KUKA KRL program: EPS_2_25694_LG02_A_20260223033040.src

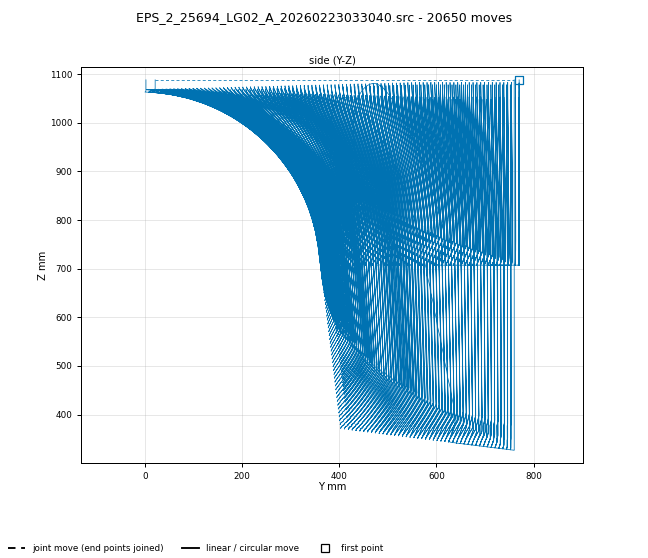
[picture p0: tool path of EPS_2_25694_LG02_A_20260223033040.src, 20650 of 20652 moves have a stored position in this frame; points joined in program order, loops and branches not executed]
&ACCESS RVP
&REL 4
&COMMENT QRS 19112012
&PARAM EDITMASK = *
DEF PART()
EXT BAS (BAS_COMMAND :IN,REAL :IN )
INT I
BAS (#INITMOV,0 )

;KUKA QRS Post kuka4.cps  Date:22-06-2017 !

File_ID=3059

QRS_PRE_INIT()

;Init var - Until changes are made in qrs_pre_init
Outlet_Square_prg=0
Inlet_1_Square_prg=0
Inlet_2_Square_prg=0
Inlet_3_Square_prg=0
Inlet_4_Square_prg=0
Inlet_5_Square_prg=0

Outlet_1={X 0.000, Y 562.000, Z 735.500, B 0.000, E1 0.000 }
Outlet_1={X 0.000, Y 562.000, Z 735.500, B 0.000, E1 0.000 }
Inlet_1={X 0.000, Y 562.000, Z 705.500, B 0.000, E1 182.000 }
Inlet_1={X 0.000, Y 562.000, Z 705.500, B 0.000, E1 182.000 }
Outlet_1_type=686
Inlet_1_type=686
Inlet_1_type=686
;QRS#1=Sidecore dimensions
;QRS#2=675-27" Concrete
;QRS#3=675-27" Concrete
;QRS#4=
;QRS#5=
;QRS#6=
;QRS#7=
;QRS#8=
;QRS#9=S306-38L
;QRS#10=S306-38L
;QRS#11=
;QRS#12=
;QRS#13=
;QRS#14=
;QRS#15=
;QRS#16=1524x152x1524 5'
;QRS#17=EPS Height
;QRS#18=1078,5
;QRS#19=*
;QRS#20= UPDATED VERSION 22-06-2017
;QRS#21=*
Outlet_Square=0550
Inlet_1_Square=0550
Inlet_2_Square=0
Inlet_3_Square=0
Inlet_4_Square=0
Inlet_5_Square=0
Mill_Square=1
Outlet_Square_Prg=265
Inlet_1_Square_prg=265
Inlet_1_Square_prg=265

QRS_INIT()

$ADVANCE=5

; T1
PTP {E1 171.77,E2 171.77}
PTP {X 0,Y 770.022,A -85,B 0,C 180,E1 171.77,E2 171.77,E3 0,E4 0,E5 0,E6 0}
QRS_SPEED_INIT()
LIN {X 0,Y 770.022,Z 1088.5,A -85,B 0,C 180,E1 171.77,E2 171.77,E3 0,E4 0,E5 0,E6 0} C_VEL
LIN {X 0,Y 770.022,Z 709.31,A -85,B 0,C 180,E1 171.77,E2 171.77} C_VEL
LIN {X 0,Y 769.965,Z 707.31,A -85,B 0,C 180,E1 171.919,E2 171.919} C_VEL
LIN {X 0,Y 770.089,Z 707.31,A -85,B 0,C 180,E1 175.346,E2 175.346} C_VEL
LIN {X 0,Y 770.137,Z 707.31,A -85,B 0,C 180,E1 180.93,E2 180.93} C_VEL
LIN {X 0,Y 770.147,Z 707.31,A -85,B 0,C 180,E1 186.522,E2 186.522} C_VEL
LIN {X 0,Y 770.143,Z 707.31,A -85,B 0,C 180,E1 190.282,E2 190.282} C_VEL
LIN {X 0,Y 769.943,Z 707.31,A -85,B 0,C 180,E1 194.091,E2 194.091} C_VEL
LIN {X 0,Y 769.516,Z 707.31,A -85,B 0,C 180,E1 196.027,E2 196.027} C_VEL
LIN {X 0,Y 770.012,Z 707.31,A -85,B 0,C 180,E1 199.927,E2 199.927} C_VEL
LIN {X 0,Y 769.316,Z 707.31,A -85,B 0,C 180,E1 202.191,E2 202.191} C_VEL
LIN {X 0,Y 769.398,Z 707.31,A -85,B 0,C 180,E1 203.958,E2 203.958} C_VEL
LIN {X 0,Y 769.902,Z 707.31,A -85,B 0,C 180,E1 205.993,E2 205.993} C_VEL
LIN {X 0,Y 769.961,Z 707.31,A -85,B 0,C 180,E1 210.209,E2 210.209} C_VEL
LIN {X 0,Y 770.093,Z 707.31,A -85,B 0,C 180,E1 210.674,E2 210.674} C_VEL
LIN {X 0,Y 769.97,Z 707.31,A -85,B 0,C 180,E1 214.616,E2 214.616} C_VEL
LIN {X 0,Y 769.539,Z 707.31,A -85,B 0,C 180,E1 217.274,E2 217.274} C_VEL
LIN {X 0,Y 769.964,Z 707.31,A -85,B 0,C 180,E1 219.272,E2 219.272} C_VEL
LIN {X 0,Y 769.757,Z 707.31,A -85,B 0,C 180,E1 220.266,E2 220.266} C_VEL
LIN {X 0,Y 769.848,Z 707.31,A -85,B 0,C 180,E1 224.269,E2 224.269} C_VEL
LIN {X 0,Y 769.688,Z 707.31,A -85,B 0,C 180,E1 225.72,E2 225.72} C_VEL
LIN {X 0,Y 769.829,Z 707.31,A -85,B 0,C 180,E1 229.727,E2 229.727} C_VEL
LIN {X 0,Y 769.876,Z 707.31,A -85,B 0,C 180,E1 230.723,E2 230.723} C_VEL
LIN {X 0,Y 769.499,Z 707.31,A -85,B 0,C 180,E1 233.066,E2 233.066} C_VEL
LIN {X 0,Y 769.922,Z 707.31,A -85,B 0,C 180,E1 235.382,E2 235.382} C_VEL
LIN {X 0,Y 770.114,Z 707.31,A -85,B 0,C 180,E1 240.252,E2 240.252} C_VEL
LIN {X 0,Y 769.925,Z 707.31,A -85,B 0,C 180,E1 240.47,E2 240.47} C_VEL
LIN {X 0,Y 768.498,Z 707.31,A -85,B 0,C 180,E1 240.635,E2 240.635} C_VEL
LIN {X 0,Y 768.109,Z 707.31,A -85,B 0,C 180,E1 240.658,E2 240.658} C_VEL
LIN {X 0,Y 769.095,Z 710.734,A -85,B 0,C 180,E1 240.752,E2 240.752} C_VEL
LIN {X 0,Y 769.603,Z 712.954,A -85,B 0,C 180,E1 240.796,E2 240.796} C_VEL
LIN {X 0,Y 769.831,Z 753.408,A -85,B 0,C 180,E1 241.229,E2 241.229} C_VEL
LIN {X 0,Y 769.934,Z 774.829,A -85,B 0,C 180,E1 241.5,E2 241.5} C_VEL
LIN {X 0,Y 769.745,Z 790.859,A -85,B 0,C 180,E1 241.76,E2 241.76} C_VEL
LIN {X 0,Y 769.973,Z 808.408,A -85,B 0,C 180,E1 242.135,E2 242.135} C_VEL
LIN {X 0,Y 769.941,Z 824.72,A -85,B 0,C 180,E1 242.54,E2 242.54} C_VEL
LIN {X 0,Y 769.833,Z 835.541,A -85,B 0,C 180,E1 242.844,E2 242.844} C_VEL
LIN {X 0,Y 769.948,Z 845.365,A -85,B 0,C 180,E1 243.157,E2 243.157} C_VEL
LIN {X 0,Y 769.988,Z 856.534,A -85,B 0,C 180,E1 243.531,E2 243.531} C_VEL
LIN {X 0,Y 769.881,Z 872.728,A -85,B 0,C 180,E1 244.138,E2 244.138} C_VEL
LIN {X 0,Y 770.005,Z 886.353,A -85,B 0,C 180,E1 244.711,E2 244.711} C_VEL
LIN {X 0,Y 769.999,Z 902.655,A -85,B 0,C 180,E1 245.473,E2 245.473} C_VEL
LIN {X 0,Y 769.936,Z 916.578,A -85,B 0,C 180,E1 246.187,E2 246.187} C_VEL
LIN {X 0,Y 769.972,Z 930.073,A -85,B 0,C 180,E1 246.948,E2 246.948} C_VEL
LIN {X 0,Y 770.004,Z 943.245,A -85,B 0,C 180,E1 247.759,E2 247.759} C_VEL
LIN {X 0,Y 770.023,Z 955.747,A -85,B 0,C 180,E1 248.596,E2 248.596} C_VEL
LIN {X 0,Y 769.988,Z 967.476,A -85,B 0,C 180,E1 249.447,E2 249.447} C_VEL
LIN {X 0,Y 769.996,Z 980.009,A -85,B 0,C 180,E1 250.443,E2 250.443} C_VEL
LIN {X 0,Y 770.035,Z 990.038,A -85,B 0,C 180,E1 251.305,E2 251.305} C_VEL
LIN {X 0,Y 769.912,Z 1001.083,A -85,B 0,C 180,E1 252.335,E2 252.335} C_VEL
LIN {X 0,Y 769.935,Z 1010.25,A -85,B 0,C 180,E1 253.265,E2 253.265} C_VEL
LIN {X 0,Y 770.052,Z 1020.333,A -85,B 0,C 180,E1 254.393,E2 254.393} C_VEL
LIN {X 0,Y 769.892,Z 1028.715,A -85,B 0,C 180,E1 255.404,E2 255.404} C_VEL
LIN {X 0,Y 769.938,Z 1037.752,A -85,B 0,C 180,E1 256.627,E2 256.627} C_VEL
LIN {X 0,Y 770.084,Z 1044.177,A -85,B 0,C 180,E1 257.583,E2 257.583} C_VEL
LIN {X 0,Y 769.904,Z 1051.422,A -85,B 0,C 180,E1 258.768,E2 258.768} C_VEL
LIN {X 0,Y 769.98,Z 1057.755,A -85,B 0,C 180,E1 259.952,E2 259.952} C_VEL
LIN {X 0,Y 770.017,Z 1062.183,A -85,B 0,C 180,E1 260.895,E2 260.895} C_VEL
LIN {X 0,Y 769.897,Z 1065.267,A -85,B 0,C 180,E1 261.6,E2 261.6} C_VEL
LIN {X 0,Y 769.889,Z 1069.496,A -85,B 0,C 180,E1 262.687,E2 262.687} C_VEL
LIN {X 0,Y 770.095,Z 1073.277,A -85,B 0,C 180,E1 263.852,E2 263.852} C_VEL
LIN {X 0,Y 769.943,Z 1075.349,A -85,B 0,C 180,E1 264.598,E2 264.598} C_VEL
LIN {X 0,Y 769.823,Z 1077.197,A -85,B 0,C 180,E1 265.344,E2 265.344} C_VEL
LIN {X 0,Y 769.892,Z 1079.406,A -85,B 0,C 180,E1 266.464,E2 266.464} C_VEL
LIN {X 0,Y 770.036,Z 1080.477,A -85,B 0,C 180,E1 267.209,E2 267.209} C_VEL
LIN {X 0,Y 769.896,Z 1081.687,A -85,B 0,C 180,E1 268.326,E2 268.326} C_VEL
LIN {X 0,Y 769.819,Z 1082.188,A -85,B 0,C 180,E1 269.07,E2 269.07} C_VEL
LIN {X 0,Y 770.094,Z 1082.112,A -85,B 0,C 180,E1 270.93,E2 270.93} C_VEL
LIN {X 0,Y 769.957,Z 1081.671,A -85,B 0,C 180,E1 271.674,E2 271.674} C_VEL
LIN {X 0,Y 769.922,Z 1080.508,A -85,B 0,C 180,E1 272.791,E2 272.791} C_VEL
LIN {X 0,Y 770.08,Z 1078.703,A -85,B 0,C 180,E1 273.908,E2 273.908} C_VEL
LIN {X 0,Y 769.95,Z 1077.164,A -85,B 0,C 180,E1 274.655,E2 274.655} C_VEL
LIN {X 0,Y 769.804,Z 1074.365,A -85,B 0,C 180,E1 275.777,E2 275.777} C_VEL
LIN {X 0,Y 769.869,Z 1072.15,A -85,B 0,C 180,E1 276.525,E2 276.525} C_VEL
LIN {X 0,Y 770.043,Z 1069.113,A -85,B 0,C 180,E1 277.415,E2 277.415} C_VEL
LIN {X 0,Y 769.819,Z 1063.335,A -85,B 0,C 180,E1 278.872,E2 278.872} C_VEL
LIN {X 0,Y 769.862,Z 1057.782,A -85,B 0,C 180,E1 280.05,E2 280.05} C_VEL
LIN {X 0,Y 770.061,Z 1051.388,A -85,B 0,C 180,E1 281.23,E2 281.23} C_VEL
LIN {X 0,Y 769.867,Z 1044.221,A -85,B 0,C 180,E1 282.42,E2 282.42} C_VEL
LIN {X 0,Y 769.93,Z 1036.081,A -85,B 0,C 180,E1 283.613,E2 283.613} C_VEL
LIN {X 0,Y 770.069,Z 1028.6,A -85,B 0,C 180,E1 284.603,E2 284.603} C_VEL
LIN {X 0,Y 769.93,Z 1018.062,A -85,B 0,C 180,E1 285.875,E2 285.875} C_VEL
LIN {X 0,Y 770.036,Z 1008.27,A -85,B 0,C 180,E1 286.937,E2 286.937} C_VEL
LIN {X 0,Y 770.027,Z 997.988,A -85,B 0,C 180,E1 287.96,E2 287.96} C_VEL
LIN {X 0,Y 769.959,Z 987.253,A -85,B 0,C 180,E1 288.942,E2 288.942} C_VEL
LIN {X 0,Y 770.039,Z 977.032,A -85,B 0,C 180,E1 289.803,E2 289.803} C_VEL
LIN {X 0,Y 770.021,Z 964.62,A -85,B 0,C 180,E1 290.763,E2 290.763} C_VEL
LIN {X 0,Y 769.992,Z 953.247,A -85,B 0,C 180,E1 291.577,E2 291.577} C_VEL
LIN {X 0,Y 770.022,Z 940.144,A -85,B 0,C 180,E1 292.436,E2 292.436} C_VEL
LIN {X 0,Y 770.026,Z 926.8,A -85,B 0,C 180,E1 293.24,E2 293.24} C_VEL
LIN {X 0,Y 769.999,Z 912.592,A -85,B 0,C 180,E1 294.022,E2 294.022} C_VEL
LIN {X 0,Y 769.954,Z 899.229,A -85,B 0,C 180,E1 294.697,E2 294.697} C_VEL
LIN {X 0,Y 770.006,Z 884.351,A -85,B 0,C 180,E1 295.375,E2 295.375} C_VEL
LIN {X 0,Y 769.96,Z 868.011,A -85,B 0,C 180,E1 296.044,E2 296.044} C_VEL
LIN {X 0,Y 769.9,Z 855.049,A -85,B 0,C 180,E1 296.527,E2 296.527} C_VEL
LIN {X 0,Y 769.996,Z 836.827,A -85,B 0,C 180,E1 297.113,E2 297.113} C_VEL
LIN {X 0,Y 769.884,Z 820.283,A -85,B 0,C 180,E1 297.579,E2 297.579} C_VEL
LIN {X 0,Y 769.807,Z 811.166,A -85,B 0,C 180,E1 297.804,E2 297.804} C_VEL
LIN {X 0,Y 769.928,Z 802.17,A -85,B 0,C 180,E1 298.003,E2 298.003} C_VEL
LIN {X 0,Y 769.948,Z 787.456,A -85,B 0,C 180,E1 298.293,E2 298.293} C_VEL
LIN {X 0,Y 769.698,Z 770.151,A -85,B 0,C 180,E1 298.575,E2 298.575} C_VEL
LIN {X 0,Y 769.766,Z 750.318,A -85,B 0,C 180,E1 298.806,E2 298.806} C_VEL
LIN {X 0,Y 769.682,Z 714.778,A -85,B 0,C 180,E1 299.181,E2 299.181} C_VEL
LIN {X 0,Y 769.131,Z 710.918,A -85,B 0,C 180,E1 299.245,E2 299.245} C_VEL
LIN {X 0,Y 767.905,Z 707.31,A -85,B 0,C 180,E1 299.334,E2 299.334} C_VEL
LIN {X 0,Y 769.925,Z 707.31,A -85,B 0,C 180,E1 299.53,E2 299.53} C_VEL
LIN {X 0,Y 770.155,Z 707.31,A -85,B 0,C 180,E1 299.746,E2 299.746} C_VEL
LIN {X 0,Y 770.109,Z 707.31,A -85,B 0,C 180,E1 300.676,E2 300.676} C_VEL
LIN {X 0,Y 769.956,Z 707.31,A -85,B 0,C 180,E1 304.616,E2 304.616} C_VEL
LIN {X 0,Y 769.531,Z 707.31,A -85,B 0,C 180,E1 307.274,E2 307.274} C_VEL
LIN {X 0,Y 769.966,Z 707.31,A -85,B 0,C 180,E1 309.271,E2 309.271} C_VEL
LIN {X 0,Y 769.769,Z 707.31,A -85,B 0,C 180,E1 310.267,E2 310.267} C_VEL
LIN {X 0,Y 769.861,Z 707.31,A -85,B 0,C 180,E1 314.268,E2 314.268} C_VEL
LIN {X 0,Y 769.694,Z 707.31,A -85,B 0,C 180,E1 315.72,E2 315.72} C_VEL
LIN {X 0,Y 769.828,Z 707.31,A -85,B 0,C 180,E1 319.727,E2 319.727} C_VEL
LIN {X 0,Y 769.883,Z 707.31,A -85,B 0,C 180,E1 320.723,E2 320.723} C_VEL
LIN {X 0,Y 769.518,Z 707.31,A -85,B 0,C 180,E1 323.067,E2 323.067} C_VEL
LIN {X 0,Y 769.966,Z 707.31,A -85,B 0,C 180,E1 325.384,E2 325.384} C_VEL
LIN {X 0,Y 770.084,Z 707.31,A -85,B 0,C 180,E1 329.327,E2 329.327} C_VEL
LIN {X 0,Y 769.954,Z 707.31,A -85,B 0,C 180,E1 329.791,E2 329.791} C_VEL
LIN {X 0,Y 769.909,Z 707.31,A -85,B 0,C 180,E1 334.007,E2 334.007} C_VEL
LIN {X 0,Y 769.391,Z 707.31,A -85,B 0,C 180,E1 336.042,E2 336.042} C_VEL
LIN {X 0,Y 769.371,Z 707.31,A -85,B 0,C 180,E1 338.063,E2 338.063} C_VEL
LIN {X 0,Y 770.006,Z 707.31,A -85,B 0,C 180,E1 340.073,E2 340.073} C_VEL
LIN {X 0,Y 769.528,Z 707.31,A -85,B 0,C 180,E1 343.974,E2 343.974} C_VEL
LIN {X 0,Y 769.936,Z 707.31,A -85,B 0,C 180,E1 345.909,E2 345.909} C_VEL
LIN {X 0,Y 770.137,Z 707.31,A -85,B 0,C 180,E1 349.718,E2 349.718} C_VEL
LIN {X 0,Y 770.151,Z 707.31,A -85,B 0,C 180,E1 353.478,E2 353.478} C_VEL
LIN {X 0,Y 770.123,Z 707.31,A -85,B 0,C 180,E1 359.07,E2 359.07} C_VEL
LIN {X 0,Y 770.092,Z 707.31,A -85,B 0,C 180,E1 364.654,E2 364.654} C_VEL
LIN {X 0,Y 770.054,Z 707.31,A -85,B 0,C 180,E1 370.283,E2 370.283} C_VEL
LIN {X 0,Y 769.882,Z 707.31,A -85,B 0,C 180,E1 374.092,E2 374.092} C_VEL
LIN {X 0,Y 769.483,Z 707.31,A -85,B 0,C 180,E1 376.027,E2 376.027} C_VEL
LIN {X 0,Y 770.04,Z 707.31,A -85,B 0,C 180,E1 379.926,E2 379.926} C_VEL
LIN {X 0,Y 769.697,Z 707.31,A -85,B 0,C 180,E1 382.261,E2 382.261} C_VEL
LIN {X 0,Y 770.058,Z 707.31,A -85,B 0,C 180,E1 383.936,E2 383.936} C_VEL
LIN {X 0,Y 769.305,Z 707.31,A -85,B 0,C 180,E1 386.69,E2 386.69} C_VEL
LIN {X 0,Y 769.438,Z 707.31,A -85,B 0,C 180,E1 388.1,E2 388.1} C_VEL
LIN {X 0,Y 769.806,Z 707.31,A -85,B 0,C 180,E1 390.216,E2 390.216} C_VEL
LIN {X 0,Y 769.886,Z 707.31,A -85,B 0,C 180,E1 394.62,E2 394.62} C_VEL
LIN {X 0,Y 769.484,Z 707.31,A -85,B 0,C 180,E1 397.269,E2 397.269} C_VEL
LIN {X 0,Y 769.902,Z 707.31,A -85,B 0,C 180,E1 399.275,E2 399.275} C_VEL
LIN {X 0,Y 769.868,Z 707.31,A -85,B 0,C 180,E1 400.276,E2 400.276} C_VEL
LIN {X 0,Y 769.855,Z 707.31,A -85,B 0,C 180,E1 404.268,E2 404.268} C_VEL
LIN {X 0,Y 769.692,Z 707.31,A -85,B 0,C 180,E1 405.72,E2 405.72} C_VEL
LIN {X 0,Y 769.873,Z 707.31,A -85,B 0,C 180,E1 409.724,E2 409.724} C_VEL
LIN {X 0,Y 770.006,Z 707.31,A -85,B 0,C 180,E1 410.731,E2 410.731} C_VEL
LIN {X 0,Y 769.993,Z 707.31,A -85,B 0,C 180,E1 413.093,E2 413.093} C_VEL
LIN {X 0,Y 769.36,Z 707.31,A -85,B 0,C 180,E1 415.936,E2 415.936} C_VEL
LIN {X 0,Y 770.019,Z 707.31,A -85,B 0,C 180,E1 418.367,E2 418.367} C_VEL
LIN {X 0,Y 769.919,Z 707.31,A -85,B 0,C 180,E1 418.779,E2 418.779} C_VEL
LIN {X 0,Y 768.954,Z 707.31,A -85,B 0,C 180,E1 418.939,E2 418.939} C_VEL
LIN {X 0,Y 768.758,Z 707.31,A -85,B 0,C 180,E1 418.958,E2 418.958} C_VEL
LIN {X 0,Y 768.921,Z 707.833,A -85,B 0,C 180,E1 418.984,E2 418.984} C_VEL
LIN {X 0,Y 769.552,Z 709.481,A -85,B 0,C 180,E1 419.027,E2 419.027} C_VEL
LIN {X 0,Y 769.707,Z 712.843,A -85,B 0,C 180,E1 419.068,E2 419.068} C_VEL
LIN {X 0,Y 769.864,Z 732.648,A -85,B 0,C 180,E1 419.294,E2 419.294} C_VEL
LIN {X 0,Y 769.85,Z 745.446,A -85,B 0,C 180,E1 419.462,E2 419.462} C_VEL
LIN {X 0,Y 769.757,Z 755.61,A -85,B 0,C 180,E1 419.624,E2 419.624} C_VEL
LIN {X 0,Y 769.862,Z 764.873,A -85,B 0,C 180,E1 419.801,E2 419.801} C_VEL
LIN {X 0,Y 769.858,Z 778.456,A -85,B 0,C 180,E1 420.086,E2 420.086} C_VEL
LIN {X 0,Y 769.821,Z 788.716,A -85,B 0,C 180,E1 420.335,E2 420.335} C_VEL
LIN {X 0,Y 769.911,Z 797.522,A -85,B 0,C 180,E1 420.574,E2 420.574} C_VEL
LIN {X 0,Y 769.941,Z 810.99,A -85,B 0,C 180,E1 420.968,E2 420.968} C_VEL
LIN {X 0,Y 769.825,Z 825.977,A -85,B 0,C 180,E1 421.459,E2 421.459} C_VEL
LIN {X 0,Y 769.962,Z 842.279,A -85,B 0,C 180,E1 422.077,E2 422.077} C_VEL
LIN {X 0,Y 769.92,Z 857.12,A -85,B 0,C 180,E1 422.698,E2 422.698} C_VEL
LIN {X 0,Y 769.996,Z 872.707,A -85,B 0,C 180,E1 423.43,E2 423.43} C_VEL
LIN {X 0,Y 770.001,Z 885.763,A -85,B 0,C 180,E1 424.099,E2 424.099} C_VEL
LIN {X 0,Y 769.962,Z 899.708,A -85,B 0,C 180,E1 424.881,E2 424.881} C_VEL
LIN {X 0,Y 769.97,Z 913.421,A -85,B 0,C 180,E1 425.725,E2 425.725} C_VEL
LIN {X 0,Y 769.995,Z 926.011,A -85,B 0,C 180,E1 426.57,E2 426.57} C_VEL
LIN {X 0,Y 770.041,Z 938.667,A -85,B 0,C 180,E1 427.497,E2 427.497} C_VEL
LIN {X 0,Y 769.962,Z 949.338,A -85,B 0,C 180,E1 428.34,E2 428.34} C_VEL
LIN {X 0,Y 769.965,Z 960.346,A -85,B 0,C 180,E1 429.286,E2 429.286} C_VEL
LIN {X 0,Y 770.061,Z 970.115,A -85,B 0,C 180,E1 430.198,E2 430.198} C_VEL
LIN {X 0,Y 769.912,Z 980.998,A -85,B 0,C 180,E1 431.302,E2 431.302} C_VEL
LIN {X 0,Y 769.954,Z 990.166,A -85,B 0,C 180,E1 432.323,E2 432.323} C_VEL
LIN {X 0,Y 770.03,Z 998.826,A -85,B 0,C 180,E1 433.38,E2 433.38} C_VEL
LIN {X 0,Y 769.876,Z 1007.704,A -85,B 0,C 180,E1 434.572,E2 434.572} C_VEL
LIN {X 0,Y 769.971,Z 1014.548,A -85,B 0,C 180,E1 435.59,E2 435.59} C_VEL
LIN {X 0,Y 770.061,Z 1019.352,A -85,B 0,C 180,E1 436.39,E2 436.39} C_VEL
LIN {X 0,Y 769.933,Z 1023.47,A -85,B 0,C 180,E1 437.104,E2 437.104} C_VEL
LIN {X 0,Y 769.882,Z 1028.518,A -85,B 0,C 180,E1 438.056,E2 438.056} C_VEL
LIN {X 0,Y 770.047,Z 1033.985,A -85,B 0,C 180,E1 439.244,E2 439.244} C_VEL
LIN {X 0,Y 769.897,Z 1037.803,A -85,B 0,C 180,E1 440.187,E2 440.187} C_VEL
LIN {X 0,Y 769.792,Z 1041.151,A -85,B 0,C 180,E1 441.128,E2 441.128} C_VEL
LIN {X 0,Y 769.817,Z 1042.735,A -85,B 0,C 180,E1 441.599,E2 441.599} C_VEL
LIN {X 0,Y 770.005,Z 1045.491,A -85,B 0,C 180,E1 442.611,E2 442.611} C_VEL
LIN {X 0,Y 769.973,Z 1047.526,A -85,B 0,C 180,E1 443.476,E2 443.476} C_VEL
LIN {X 0,Y 769.865,Z 1049.125,A -85,B 0,C 180,E1 444.224,E2 444.224} C_VEL
LIN {X 0,Y 769.912,Z 1050.786,A -85,B 0,C 180,E1 445.345,E2 445.345} C_VEL
LIN {X 0,Y 770.059,Z 1051.473,A -85,B 0,C 180,E1 446.092,E2 446.092} C_VEL
LIN {X 0,Y 769.847,Z 1052.232,A -85,B 0,C 180,E1 447.209,E2 447.209} C_VEL
LIN {X 0,Y 769.868,Z 1052.125,A -85,B 0,C 180,E1 449.07,E2 449.07} C_VEL
LIN {X 0,Y 770.051,Z 1051.152,A -85,B 0,C 180,E1 450.186,E2 450.186} C_VEL
LIN {X 0,Y 769.859,Z 1049.146,A -85,B 0,C 180,E1 451.674,E2 451.674} C_VEL
LIN {X 0,Y 769.988,Z 1046.777,A -85,B 0,C 180,E1 452.791,E2 452.791} C_VEL
LIN {X 0,Y 770.031,Z 1044.835,A -85,B 0,C 180,E1 453.536,E2 453.536} C_VEL
LIN {X 0,Y 769.875,Z 1042.817,A -85,B 0,C 180,E1 454.282,E2 454.282} C_VEL
LIN {X 0,Y 769.825,Z 1039.065,A -85,B 0,C 180,E1 455.403,E2 455.403} C_VEL
LIN {X 0,Y 770.076,Z 1033.466,A -85,B 0,C 180,E1 456.783,E2 456.783} C_VEL
LIN {X 0,Y 769.835,Z 1027.352,A -85,B 0,C 180,E1 458.086,E2 458.086} C_VEL
LIN {X 0,Y 769.838,Z 1021.898,A -85,B 0,C 180,E1 459.107,E2 459.107} C_VEL
LIN {X 0,Y 770.077,Z 1014.746,A -85,B 0,C 180,E1 460.283,E2 460.283} C_VEL
LIN {X 0,Y 769.892,Z 1006.814,A -85,B 0,C 180,E1 461.469,E2 461.469} C_VEL
LIN {X 0,Y 769.88,Z 997.877,A -85,B 0,C 180,E1 462.658,E2 462.658} C_VEL
LIN {X 0,Y 770.052,Z 987.84,A -85,B 0,C 180,E1 463.85,E2 463.85} C_VEL
LIN {X 0,Y 769.933,Z 979.058,A -85,B 0,C 180,E1 464.816,E2 464.816} C_VEL
LIN {X 0,Y 769.965,Z 967.997,A -85,B 0,C 180,E1 465.917,E2 465.917} C_VEL
LIN {X 0,Y 770.065,Z 958.104,A -85,B 0,C 180,E1 466.822,E2 466.822} C_VEL
LIN {X 0,Y 769.962,Z 946.275,A -85,B 0,C 180,E1 467.819,E2 467.819} C_VEL
LIN {X 0,Y 769.979,Z 934.941,A -85,B 0,C 180,E1 468.696,E2 468.696} C_VEL
LIN {X 0,Y 770.027,Z 922.862,A -85,B 0,C 180,E1 469.556,E2 469.556} C_VEL
LIN {X 0,Y 769.986,Z 910.109,A -85,B 0,C 180,E1 470.394,E2 470.394} C_VEL
LIN {X 0,Y 770.004,Z 897.682,A -85,B 0,C 180,E1 471.146,E2 471.146} C_VEL
LIN {X 0,Y 769.988,Z 883.743,A -85,B 0,C 180,E1 471.919,E2 471.919} C_VEL
LIN {X 0,Y 770.021,Z 869.346,A -85,B 0,C 180,E1 472.644,E2 472.644} C_VEL
LIN {X 0,Y 769.963,Z 853.47,A -85,B 0,C 180,E1 473.368,E2 473.368} C_VEL
LIN {X 0,Y 769.996,Z 838.489,A -85,B 0,C 180,E1 473.98,E2 473.98} C_VEL
LIN {X 0,Y 770.007,Z 823.517,A -85,B 0,C 180,E1 474.529,E2 474.529} C_VEL
LIN {X 0,Y 769.806,Z 806.359,A -85,B 0,C 180,E1 475.088,E2 475.088} C_VEL
LIN {X 0,Y 769.958,Z 790.171,A -85,B 0,C 180,E1 475.534,E2 475.534} C_VEL
LIN {X 0,Y 769.914,Z 773.708,A -85,B 0,C 180,E1 475.927,E2 475.927} C_VEL
LIN {X 0,Y 769.78,Z 761.942,A -85,B 0,C 180,E1 476.172,E2 476.172} C_VEL
LIN {X 0,Y 769.993,Z 742.231,A -85,B 0,C 180,E1 476.493,E2 476.493} C_VEL
LIN {X 0,Y 769.805,Z 720.28,A -85,B 0,C 180,E1 476.76,E2 476.76} C_VEL
LIN {X 0,Y 769.598,Z 707.31,A -85,B 0,C 180,E1 476.907,E2 476.907} C_VEL
LIN {X 0,Y 770.053,Z 707.31,A -85,B 0,C 180,E1 476.99,E2 476.99} C_VEL
LIN {X 0,Y 770.045,Z 707.31,A -85,B 0,C 180,E1 477.71,E2 477.71} C_VEL
LIN {X 0,Y 769.87,Z 707.31,A -85,B 0,C 180,E1 480.213,E2 480.213} C_VEL
LIN {X 0,Y 769.911,Z 707.31,A -85,B 0,C 180,E1 484.619,E2 484.619} C_VEL
LIN {X 0,Y 769.501,Z 707.31,A -85,B 0,C 180,E1 487.271,E2 487.271} C_VEL
LIN {X 0,Y 769.942,Z 707.31,A -85,B 0,C 180,E1 489.273,E2 489.273} C_VEL
LIN {X 0,Y 769.884,Z 707.31,A -85,B 0,C 180,E1 490.277,E2 490.277} C_VEL
LIN {X 0,Y 769.697,Z 707.31,A -85,B 0,C 180,E1 494.28,E2 494.28} C_VEL
LIN {X 0,Y 769.864,Z 707.31,A -85,B 0,C 180,E1 495.732,E2 495.732} C_VEL
LIN {X 0,Y 769.869,Z 707.31,A -85,B 0,C 180,E1 499.724,E2 499.724} C_VEL
LIN {X 0,Y 769.895,Z 707.31,A -85,B 0,C 180,E1 500.724,E2 500.724} C_VEL
LIN {X 0,Y 769.494,Z 707.31,A -85,B 0,C 180,E1 503.065,E2 503.065} C_VEL
LIN {X 0,Y 769.937,Z 707.31,A -85,B 0,C 180,E1 505.382,E2 505.382} C_VEL
LIN {X 0,Y 770.095,Z 707.31,A -85,B 0,C 180,E1 509.326,E2 509.326} C_VEL
LIN {X 0,Y 769.421,Z 707.31,A -85,B 0,C 180,E1 511.899,E2 511.899} C_VEL
LIN {X 0,Y 769.915,Z 707.31,A -85,B 0,C 180,E1 514.007,E2 514.007} C_VEL
LIN {X 0,Y 769.418,Z 707.31,A -85,B 0,C 180,E1 516.043,E2 516.043} C_VEL
LIN {X 0,Y 769.396,Z 707.31,A -85,B 0,C 180,E1 518.063,E2 518.063} C_VEL
LIN {X 0,Y 770.045,Z 707.31,A -85,B 0,C 180,E1 520.074,E2 520.074} C_VEL
LIN {X 0,Y 769.472,Z 707.31,A -85,B 0,C 180,E1 523.973,E2 523.973} C_VEL
LIN {X 0,Y 770.019,Z 707.31,A -85,B 0,C 180,E1 525.91,E2 525.91} C_VEL
LIN {X 0,Y 770.104,Z 707.31,A -85,B 0,C 180,E1 527.821,E2 527.821} C_VEL
LIN {X 0,Y 770.094,Z 707.31,A -85,B 0,C 180,E1 531.602,E2 531.602} C_VEL
LIN {X 0,Y 769.965,Z 707.31,A -85,B 0,C 180,E1 531.919,E2 531.919} C_VEL
LIN {X 0,Y 765.777,Z 707.31,A -85,B 0,C 180,E1 533.187,E2 533.187} C_VEL
LIN {X 0,Y 761.897,Z 707.31,A -85,B 0,C 180,E1 534.468,E2 534.468} C_VEL
LIN {X 0,Y 762.122,Z 707.31,A -85,B 0,C 180,E1 541.137,E2 541.137} C_VEL
LIN {X 0,Y 762.14,Z 707.31,A -85,B 0,C 180,E1 546.85,E2 546.85} C_VEL
LIN {X 0,Y 761.837,Z 707.31,A -85,B 0,C 180,E1 551.471,E2 551.471} C_VEL
LIN {X 0,Y 761.759,Z 707.31,A -85,B 0,C 180,E1 554.986,E2 554.986} C_VEL
LIN {X 0,Y 762.04,Z 707.31,A -85,B 0,C 180,E1 559.756,E2 559.756} C_VEL
LIN {X 0,Y 761.797,Z 707.31,A -85,B 0,C 180,E1 566.47,E2 566.47} C_VEL
LIN {X 0,Y 761.973,Z 707.31,A -85,B 0,C 180,E1 571.22,E2 571.22} C_VEL
LIN {X 0,Y 761.795,Z 707.31,A -85,B 0,C 180,E1 575.353,E2 575.353} C_VEL
LIN {X 0,Y 762.007,Z 707.31,A -85,B 0,C 180,E1 579.519,E2 579.519} C_VEL
LIN {X 0,Y 761.959,Z 707.31,A -85,B 0,C 180,E1 584.276,E2 584.276} C_VEL
LIN {X 0,Y 761.933,Z 707.31,A -85,B 0,C 180,E1 590.861,E2 590.861} C_VEL
LIN {X 0,Y 761.696,Z 707.31,A -85,B 0,C 180,E1 596.147,E2 596.147} C_VEL
LIN {X 0,Y 761.654,Z 707.31,A -85,B 0,C 180,E1 600.317,E2 600.317} C_VEL
LIN {X 0,Y 762.123,Z 712.337,A -85,B 0,C 180,E1 600.475,E2 600.475} C_VEL
LIN {X 0,Y 762.839,Z 786.85,A -85,B 0,C 180,E1 601.409,E2 601.409} C_VEL
LIN {X 0,Y 762.789,Z 832.67,A -85,B 0,C 180,E1 602.49,E2 602.49} C_VEL
LIN {X 0,Y 762.644,Z 876.024,A -85,B 0,C 180,E1 604.012,E2 604.012} C_VEL
LIN {X 0,Y 762.508,Z 917.78,A -85,B 0,C 180,E1 606.008,E2 606.008} C_VEL
LIN {X 0,Y 762.44,Z 956.472,A -85,B 0,C 180,E1 608.426,E2 608.426} C_VEL
LIN {X 0,Y 762.326,Z 990.608,A -85,B 0,C 180,E1 611.153,E2 611.153} C_VEL
LIN {X 0,Y 762.3,Z 1021.09,A -85,B 0,C 180,E1 614.284,E2 614.284} C_VEL
LIN {X 0,Y 762.278,Z 1046.013,A -85,B 0,C 180,E1 617.66,E2 617.66} C_VEL
LIN {X 0,Y 762.152,Z 1064.516,A -85,B 0,C 180,E1 621.135,E2 621.135} C_VEL
LIN {X 0,Y 762.179,Z 1075.63,A -85,B 0,C 180,E1 624.294,E2 624.294} C_VEL
LIN {X 0,Y 762.145,Z 1082.219,A -85,B 0,C 180,E1 627.72,E2 627.72} C_VEL
LIN {X 0,Y 762.233,Z 1083.17,A -85,B 0,C 180,E1 631.139,E2 631.139} C_VEL
LIN {X 0,Y 762.137,Z 1078.459,A -85,B 0,C 180,E1 634.561,E2 634.561} C_VEL
LIN {X 0,Y 762.103,Z 1068.014,A -85,B 0,C 180,E1 638,E2 638} C_VEL
LIN {X 0,Y 762.226,Z 1052.973,A -85,B 0,C 180,E1 641.177,E2 641.177} C_VEL
LIN {X 0,Y 762.303,Z 1029.54,A -85,B 0,C 180,E1 644.682,E2 644.682} C_VEL
LIN {X 0,Y 762.302,Z 1000.259,A -85,B 0,C 180,E1 647.945,E2 647.945} C_VEL
LIN {X 0,Y 762.412,Z 965.587,A -85,B 0,C 180,E1 650.91,E2 650.91} C_VEL
LIN {X 0,Y 762.559,Z 927.911,A -85,B 0,C 180,E1 653.418,E2 653.418} C_VEL
LIN {X 0,Y 762.713,Z 885.128,A -85,B 0,C 180,E1 655.603,E2 655.603} C_VEL
LIN {X 0,Y 762.881,Z 839.545,A -85,B 0,C 180,E1 657.305,E2 657.305} C_VEL
LIN {X 0,Y 762.975,Z 795.03,A -85,B 0,C 180,E1 658.428,E2 658.428} C_VEL
LIN {X 0,Y 762.839,Z 750.718,A -85,B 0,C 180,E1 659.089,E2 659.089} C_VEL
LIN {X 0,Y 762.065,Z 712.331,A -85,B 0,C 180,E1 659.527,E2 659.527} C_VEL
LIN {X 0,Y 761.246,Z 707.31,A -85,B 0,C 180,E1 659.651,E2 659.651} C_VEL
LIN {X 0,Y 762.267,Z 707.31,A -85,B 0,C 180,E1 659.801,E2 659.801} C_VEL
LIN {X 0,Y 761.798,Z 707.31,A -85,B 0,C 180,E1 665.359,E2 665.359} C_VEL
LIN {X 0,Y 762.009,Z 707.31,A -85,B 0,C 180,E1 669.522,E2 669.522} C_VEL
LIN {X 0,Y 761.973,Z 707.31,A -85,B 0,C 180,E1 674.282,E2 674.282} C_VEL
LIN {X 0,Y 761.939,Z 707.31,A -85,B 0,C 180,E1 680.864,E2 680.864} C_VEL
LIN {X 0,Y 761.801,Z 707.31,A -85,B 0,C 180,E1 686.155,E2 686.155} C_VEL
LIN {X 0,Y 761.889,Z 707.31,A -85,B 0,C 180,E1 690.185,E2 690.185} C_VEL
LIN {X 0,Y 761.983,Z 707.31,A -85,B 0,C 180,E1 694.056,E2 694.056} C_VEL
LIN {X 0,Y 762.007,Z 707.31,A -85,B 0,C 180,E1 700.243,E2 700.243} C_VEL
LIN {X 0,Y 761.957,Z 707.31,A -85,B 0,C 180,E1 706.195,E2 706.195} C_VEL
LIN {X 0,Y 761.898,Z 707.31,A -85,B 0,C 180,E1 710.846,E2 710.846} C_VEL
LIN {X 0,Y 761.786,Z 707.31,A -85,B 0,C 180,E1 714.294,E2 714.294} C_VEL
LIN {X 0,Y 762.089,Z 707.31,A -85,B 0,C 180,E1 718.863,E2 718.863} C_VEL
LIN {X 0,Y 762.146,Z 707.31,A -85,B 0,C 180,E1 724.564,E2 724.564} C_VEL
LIN {X 0,Y 762.151,Z 707.31,A -85,B 0,C 180,E1 730.31,E2 730.31} C_VEL
LIN {X 0,Y 761.701,Z 707.31,A -85,B 0,C 180,E1 734.991,E2 734.991} C_VEL
LIN {X 0,Y 761.885,Z 707.31,A -85,B 0,C 180,E1 740.8,E2 740.8} C_VEL
LIN {X 0,Y 761.782,Z 707.31,A -85,B 0,C 180,E1 744.695,E2 744.695} C_VEL
LIN {X 0,Y 761.782,Z 707.31,A -85,B 0,C 180,E1 749.825,E2 749.825} C_VEL
LIN {X 0,Y 761.721,Z 707.31,A -85,B 0,C 180,E1 755.347,E2 755.347} C_VEL
LIN {X 0,Y 762,Z 707.31,A -85,B 0,C 180,E1 759.525,E2 759.525} C_VEL
LIN {X 0,Y 761.967,Z 707.31,A -85,B 0,C 180,E1 764.278,E2 764.278} C_VEL
LIN {X 0,Y 762.079,Z 707.31,A -85,B 0,C 180,E1 770.854,E2 770.854} C_VEL
LIN {X 0,Y 761.514,Z 707.31,A -85,B 0,C 180,E1 774.754,E2 774.754} C_VEL
LIN {X 0,Y 761.814,Z 707.31,A -85,B 0,C 180,E1 778.68,E2 778.68} C_VEL
LIN {X 0,Y 762.938,Z 739.466,A -85,B 0,C 180,E1 779.094,E2 779.094} C_VEL
LIN {X 0,Y 762.785,Z 783.666,A -85,B 0,C 180,E1 779.934,E2 779.934} C_VEL
LIN {X 0,Y 762.625,Z 828.536,A -85,B 0,C 180,E1 781.285,E2 781.285} C_VEL
LIN {X 0,Y 762.657,Z 871.502,A -85,B 0,C 180,E1 783.116,E2 783.116} C_VEL
LIN {X 0,Y 762.44,Z 912.855,A -85,B 0,C 180,E1 785.455,E2 785.455} C_VEL
LIN {X 0,Y 762.334,Z 949.172,A -85,B 0,C 180,E1 788.117,E2 788.117} C_VEL
LIN {X 0,Y 762.191,Z 981.412,A -85,B 0,C 180,E1 791.151,E2 791.151} C_VEL
LIN {X 0,Y 762.1,Z 1007.099,A -85,B 0,C 180,E1 794.281,E2 794.281} C_VEL
LIN {X 0,Y 762.081,Z 1027.671,A -85,B 0,C 180,E1 797.658,E2 797.658} C_VEL
LIN {X 0,Y 762.005,Z 1041.297,A -85,B 0,C 180,E1 800.846,E2 800.846} C_VEL
LIN {X 0,Y 762.073,Z 1049.465,A -85,B 0,C 180,E1 803.872,E2 803.872} C_VEL
LIN {X 0,Y 762.126,Z 1053.024,A -85,B 0,C 180,E1 806.581,E2 806.581} C_VEL
LIN {X 0,Y 762.177,Z 1052.427,A -85,B 0,C 180,E1 810.001,E2 810.001} C_VEL
LIN {X 0,Y 762.21,Z 1046.286,A -85,B 0,C 180,E1 813.42,E2 813.42} C_VEL
LIN {X 0,Y 762.276,Z 1034.363,A -85,B 0,C 180,E1 816.851,E2 816.851} C_VEL
LIN {X 0,Y 762.275,Z 1015.941,A -85,B 0,C 180,E1 820.307,E2 820.307} C_VEL
LIN {X 0,Y 762.227,Z 991.64,A -85,B 0,C 180,E1 823.605,E2 823.605} C_VEL
LIN {X 0,Y 762.32,Z 962.721,A -85,B 0,C 180,E1 826.605,E2 826.605} C_VEL
LIN {X 0,Y 762.393,Z 929.673,A -85,B 0,C 180,E1 829.297,E2 829.297} C_VEL
LIN {X 0,Y 762.539,Z 893.05,A -85,B 0,C 180,E1 831.648,E2 831.648} C_VEL
LIN {X 0,Y 762.704,Z 852.297,A -85,B 0,C 180,E1 833.677,E2 833.677} C_VEL
LIN {X 0,Y 762.699,Z 807.525,A -85,B 0,C 180,E1 835.329,E2 835.329} C_VEL
LIN {X 0,Y 762.875,Z 759.589,A -85,B 0,C 180,E1 836.498,E2 836.498} C_VEL
LIN {X 0,Y 762.154,Z 707.31,A -85,B 0,C 180,E1 837.214,E2 837.214} C_VEL
LIN {X 0,Y 761.597,Z 707.31,A -85,B 0,C 180,E1 841.171,E2 841.171} C_VEL
LIN {X 0,Y 761.747,Z 707.31,A -85,B 0,C 180,E1 845.346,E2 845.346} C_VEL
LIN {X 0,Y 762.032,Z 707.31,A -85,B 0,C 180,E1 849.522,E2 849.522} C_VEL
LIN {X 0,Y 761.9,Z 707.31,A -85,B 0,C 180,E1 855.88,E2 855.88} C_VEL
LIN {X 0,Y 761.948,Z 707.31,A -85,B 0,C 180,E1 860.865,E2 860.865} C_VEL
LIN {X 0,Y 761.812,Z 707.31,A -85,B 0,C 180,E1 866.151,E2 866.151} C_VEL
LIN {X 0,Y 761.818,Z 707.31,A -85,B 0,C 180,E1 870.177,E2 870.177} C_VEL
LIN {X 0,Y 762.012,Z 707.31,A -85,B 0,C 180,E1 874.053,E2 874.053} C_VEL
LIN {X 0,Y 762.071,Z 707.31,A -85,B 0,C 180,E1 880.24,E2 880.24} C_VEL
LIN {X 0,Y 762.083,Z 707.31,A -85,B 0,C 180,E1 887,E2 887} C_VEL
LIN {X 0,Y 762.055,Z 707.31,A -85,B 0,C 180,E1 891.996,E2 891.996} C_VEL
LIN {X 0,Y 761.897,Z 707.31,A -85,B 0,C 180,E1 894.468,E2 894.468} C_VEL
LIN {X 0,Y 757.871,Z 707.31,A -85,B 0,C 180,E1 895.749,E2 895.749} C_VEL
LIN {X 0,Y 753.571,Z 707.31,A -85,B 0,C 180,E1 897.044,E2 897.044} C_VEL
LIN {X 0,Y 754.208,Z 707.31,A -85,B 0,C 180,E1 901.149,E2 901.149} C_VEL
LIN {X 0,Y 754.212,Z 707.31,A -85,B 0,C 180,E1 906.922,E2 906.922} C_VEL
LIN {X 0,Y 753.911,Z 707.31,A -85,B 0,C 180,E1 911.593,E2 911.593} C_VEL
LIN {X 0,Y 753.818,Z 707.31,A -85,B 0,C 180,E1 915.214,E2 915.214} C_VEL
LIN {X 0,Y 754.063,Z 707.31,A -85,B 0,C 180,E1 919.974,E2 919.974} C_VEL
LIN {X 0,Y 753.985,Z 707.31,A -85,B 0,C 180,E1 926.24,E2 926.24} C_VEL
LIN {X 0,Y 753.992,Z 707.31,A -85,B 0,C 180,E1 931.501,E2 931.501} C_VEL
LIN {X 0,Y 753.708,Z 707.31,A -85,B 0,C 180,E1 936.463,E2 936.463} C_VEL
LIN {X 0,Y 753.866,Z 707.31,A -85,B 0,C 180,E1 940.193,E2 940.193} C_VEL
LIN {X 0,Y 753.912,Z 707.31,A -85,B 0,C 180,E1 945.29,E2 945.29} C_VEL
LIN {X 0,Y 753.913,Z 707.31,A -85,B 0,C 180,E1 949.967,E2 949.967} C_VEL
LIN {X 0,Y 753.778,Z 707.31,A -85,B 0,C 180,E1 955.742,E2 955.742} C_VEL
LIN {X 0,Y 754.219,Z 707.31,A -85,B 0,C 180,E1 960.068,E2 960.068} C_VEL
LIN {X 0,Y 755.877,Z 722.616,A -85,B 0,C 180,E1 960.317,E2 960.317} C_VEL
LIN {X 0,Y 755.858,Z 789.553,A -85,B 0,C 180,E1 961.166,E2 961.166} C_VEL
LIN {X 0,Y 755.632,Z 838.054,A -85,B 0,C 180,E1 962.364,E2 962.364} C_VEL
LIN {X 0,Y 755.415,Z 885.307,A -85,B 0,C 180,E1 964.139,E2 964.139} C_VEL
LIN {X 0,Y 755.055,Z 929.178,A -85,B 0,C 180,E1 966.41,E2 966.41} C_VEL
LIN {X 0,Y 754.764,Z 967.337,A -85,B 0,C 180,E1 969.001,E2 969.001} C_VEL
LIN {X 0,Y 754.506,Z 1000.243,A -85,B 0,C 180,E1 971.861,E2 971.861} C_VEL
LIN {X 0,Y 754.31,Z 1029.534,A -85,B 0,C 180,E1 975.158,E2 975.158} C_VEL
LIN {X 0,Y 754.251,Z 1051.274,A -85,B 0,C 180,E1 978.409,E2 978.409} C_VEL
LIN {X 0,Y 754.205,Z 1066.858,A -85,B 0,C 180,E1 981.623,E2 981.623} C_VEL
LIN {X 0,Y 754.216,Z 1077.191,A -85,B 0,C 180,E1 984.812,E2 984.812} C_VEL
LIN {X 0,Y 754.241,Z 1082.219,A -85,B 0,C 180,E1 987.697,E2 987.697} C_VEL
LIN {X 0,Y 754.33,Z 1083.171,A -85,B 0,C 180,E1 991.151,E2 991.151} C_VEL
LIN {X 0,Y 754.228,Z 1078.459,A -85,B 0,C 180,E1 994.609,E2 994.609} C_VEL
LIN {X 0,Y 754.193,Z 1068.014,A -85,B 0,C 180,E1 998.085,E2 998.085} C_VEL
LIN {X 0,Y 754.347,Z 1052.974,A -85,B 0,C 180,E1 1001.295,E2 1001.295} C_VEL
LIN {X 0,Y 754.455,Z 1029.542,A -85,B 0,C 180,E1 1004.838,E2 1004.838} C_VEL
LIN {X 0,Y 754.575,Z 1000.254,A -85,B 0,C 180,E1 1008.136,E2 1008.136} C_VEL
LIN {X 0,Y 754.806,Z 965.588,A -85,B 0,C 180,E1 1011.131,E2 1011.131} C_VEL
LIN {X 0,Y 755.129,Z 927.914,A -85,B 0,C 180,E1 1013.663,E2 1013.663} C_VEL
LIN {X 0,Y 755.446,Z 885.349,A -85,B 0,C 180,E1 1015.858,E2 1015.858} C_VEL
LIN {X 0,Y 755.764,Z 840.029,A -85,B 0,C 180,E1 1017.568,E2 1017.568} C_VEL
LIN {X 0,Y 755.993,Z 795.724,A -85,B 0,C 180,E1 1018.7,E2 1018.7} C_VEL
LIN {X 0,Y 755.957,Z 752.369,A -85,B 0,C 180,E1 1019.362,E2 1019.362} C_VEL
LIN {X 0,Y 755.1,Z 714.015,A -85,B 0,C 180,E1 1019.809,E2 1019.809} C_VEL
LIN {X 0,Y 754.332,Z 707.31,A -85,B 0,C 180,E1 1019.968,E2 1019.968} C_VEL
LIN {X 0,Y 753.816,Z 707.31,A -85,B 0,C 180,E1 1025.66,E2 1025.66} C_VEL
LIN {X 0,Y 753.873,Z 707.31,A -85,B 0,C 180,E1 1030.199,E2 1030.199} C_VEL
LIN {X 0,Y 753.919,Z 707.31,A -85,B 0,C 180,E1 1035.294,E2 1035.294} C_VEL
LIN {X 0,Y 753.918,Z 707.31,A -85,B 0,C 180,E1 1039.972,E2 1039.972} C_VEL
LIN {X 0,Y 753.865,Z 707.31,A -85,B 0,C 180,E1 1045.75,E2 1045.75} C_VEL
LIN {X 0,Y 753.981,Z 707.31,A -85,B 0,C 180,E1 1049.84,E2 1049.84} C_VEL
LIN {X 0,Y 753.728,Z 707.31,A -85,B 0,C 180,E1 1055.028,E2 1055.028} C_VEL
LIN {X 0,Y 753.857,Z 707.31,A -85,B 0,C 180,E1 1060.871,E2 1060.871} C_VEL
LIN {X 0,Y 754.012,Z 707.31,A -85,B 0,C 180,E1 1066.047,E2 1066.047} C_VEL
LIN {X 0,Y 754.014,Z 707.31,A -85,B 0,C 180,E1 1070.75,E2 1070.75} C_VEL
LIN {X 0,Y 753.928,Z 707.31,A -85,B 0,C 180,E1 1074.234,E2 1074.234} C_VEL
LIN {X 0,Y 754.175,Z 707.31,A -85,B 0,C 180,E1 1078.851,E2 1078.851} C_VEL
LIN {X 0,Y 754.212,Z 707.31,A -85,B 0,C 180,E1 1084.612,E2 1084.612} C_VEL
LIN {X 0,Y 754.197,Z 707.31,A -85,B 0,C 180,E1 1090.42,E2 1090.42} C_VEL
LIN {X 0,Y 753.751,Z 707.31,A -85,B 0,C 180,E1 1095.2,E2 1095.2} C_VEL
LIN {X 0,Y 754.101,Z 707.31,A -85,B 0,C 180,E1 1099.978,E2 1099.978} C_VEL
LIN {X 0,Y 754.175,Z 707.31,A -85,B 0,C 180,E1 1103.697,E2 1103.697} C_VEL
LIN {X 0,Y 753.797,Z 707.31,A -85,B 0,C 180,E1 1110.181,E2 1110.181} C_VEL
LIN {X 0,Y 753.745,Z 707.31,A -85,B 0,C 180,E1 1115.667,E2 1115.667} C_VEL
LIN {X 0,Y 753.923,Z 707.31,A -85,B 0,C 180,E1 1120.2,E2 1120.2} C_VEL
LIN {X 0,Y 753.917,Z 707.31,A -85,B 0,C 180,E1 1125.291,E2 1125.291} C_VEL
LIN {X 0,Y 754.071,Z 707.31,A -85,B 0,C 180,E1 1131.608,E2 1131.608} C_VEL
LIN {X 0,Y 753.728,Z 707.31,A -85,B 0,C 180,E1 1137.123,E2 1137.123} C_VEL
LIN {X 0,Y 754.18,Z 707.31,A -85,B 0,C 180,E1 1138.351,E2 1138.351} C_VEL
LIN {X 0,Y 755.942,Z 718.996,A -85,B 0,C 180,E1 1138.557,E2 1138.557} C_VEL
LIN {X 0,Y 755.881,Z 765.457,A -85,B 0,C 180,E1 1139.245,E2 1139.245} C_VEL
LIN {X 0,Y 755.727,Z 809.818,A -85,B 0,C 180,E1 1140.379,E2 1140.379} C_VEL
LIN {X 0,Y 755.407,Z 854.961,A -85,B 0,C 180,E1 1142.079,E2 1142.079} C_VEL
LIN {X 0,Y 755.085,Z 898.214,A -85,B 0,C 180,E1 1144.308,E2 1144.308} C_VEL
LIN {X 0,Y 754.814,Z 937.295,A -85,B 0,C 180,E1 1146.954,E2 1146.954} C_VEL
LIN {X 0,Y 754.585,Z 971.141,A -85,B 0,C 180,E1 1149.91,E2 1149.91} C_VEL
LIN {X 0,Y 754.438,Z 999.469,A -85,B 0,C 180,E1 1153.107,E2 1153.107} C_VEL
LIN {X 0,Y 754.332,Z 1022.918,A -85,B 0,C 180,E1 1156.649,E2 1156.649} C_VEL
LIN {X 0,Y 754.212,Z 1038.2,A -85,B 0,C 180,E1 1159.917,E2 1159.917} C_VEL
LIN {X 0,Y 754.282,Z 1047.899,A -85,B 0,C 180,E1 1163.077,E2 1163.077} C_VEL
LIN {X 0,Y 754.225,Z 1053.005,A -85,B 0,C 180,E1 1166.545,E2 1166.545} C_VEL
LIN {X 0,Y 754.277,Z 1052.446,A -85,B 0,C 180,E1 1170.001,E2 1170.001} C_VEL
LIN {X 0,Y 754.334,Z 1046.344,A -85,B 0,C 180,E1 1173.456,E2 1173.456} C_VEL
LIN {X 0,Y 754.363,Z 1034.464,A -85,B 0,C 180,E1 1176.923,E2 1176.923} C_VEL
LIN {X 0,Y 754.404,Z 1016.075,A -85,B 0,C 180,E1 1180.416,E2 1180.416} C_VEL
LIN {X 0,Y 754.437,Z 991.833,A -85,B 0,C 180,E1 1183.748,E2 1183.748} C_VEL
LIN {X 0,Y 754.616,Z 963.246,A -85,B 0,C 180,E1 1186.753,E2 1186.753} C_VEL
LIN {X 0,Y 754.825,Z 930.606,A -85,B 0,C 180,E1 1189.453,E2 1189.453} C_VEL
LIN {X 0,Y 755.123,Z 893.467,A -85,B 0,C 180,E1 1191.871,E2 1191.871} C_VEL
LIN {X 0,Y 755.438,Z 852.955,A -85,B 0,C 180,E1 1193.915,E2 1193.915} C_VEL
LIN {X 0,Y 755.602,Z 807.775,A -85,B 0,C 180,E1 1195.601,E2 1195.601} C_VEL
LIN {X 0,Y 755.895,Z 760.769,A -85,B 0,C 180,E1 1196.762,E2 1196.762} C_VEL
LIN {X 0,Y 755.113,Z 710.992,A -85,B 0,C 180,E1 1197.474,E2 1197.474} C_VEL
LIN {X 0,Y 754.145,Z 707.31,A -85,B 0,C 180,E1 1197.606,E2 1197.606} C_VEL
LIN {X 0,Y 753.593,Z 707.31,A -85,B 0,C 180,E1 1202.885,E2 1202.885} C_VEL
LIN {X 0,Y 753.7,Z 707.31,A -85,B 0,C 180,E1 1207.099,E2 1207.099} C_VEL
LIN {X 0,Y 753.62,Z 707.31,A -85,B 0,C 180,E1 1211.574,E2 1211.574} C_VEL
LIN {X 0,Y 753.836,Z 707.31,A -85,B 0,C 180,E1 1216.361,E2 1216.361} C_VEL
LIN {X 0,Y 753.839,Z 707.31,A -85,B 0,C 180,E1 1221.629,E2 1221.629} C_VEL
LIN {X 0,Y 753.862,Z 707.31,A -85,B 0,C 180,E1 1225.745,E2 1225.745} C_VEL
LIN {X 0,Y 753.94,Z 707.31,A -85,B 0,C 180,E1 1229.833,E2 1229.833} C_VEL
LIN {X 0,Y 753.772,Z 707.31,A -85,B 0,C 180,E1 1235.025,E2 1235.025} C_VEL
LIN {X 0,Y 753.857,Z 707.31,A -85,B 0,C 180,E1 1240.874,E2 1240.874} C_VEL
LIN {X 0,Y 754.21,Z 707.31,A -85,B 0,C 180,E1 1247.229,E2 1247.229} C_VEL
LIN {X 0,Y 754.137,Z 707.31,A -85,B 0,C 180,E1 1251.914,E2 1251.914} C_VEL
LIN {X 0,Y 753.738,Z 707.31,A -85,B 0,C 180,E1 1256.54,E2 1256.54} C_VEL
LIN {X 0,Y 753.571,Z 707.31,A -85,B 0,C 180,E1 1257.044,E2 1257.044} C_VEL
LIN {X 0,Y 749.478,Z 707.31,A -85,B 0,C 180,E1 1258.341,E2 1258.341} C_VEL
LIN {X 0,Y 745.8,Z 707.31,A -85,B 0,C 180,E1 1259.652,E2 1259.652} C_VEL
LIN {X 0,Y 745.783,Z 707.31,A -85,B 0,C 180,E1 1262.327,E2 1262.327} C_VEL
LIN {X 0,Y 746.29,Z 707.31,A -85,B 0,C 180,E1 1266.996,E2 1266.996} C_VEL
LIN {X 0,Y 745.989,Z 707.31,A -85,B 0,C 180,E1 1271.718,E2 1271.718} C_VEL
LIN {X 0,Y 745.91,Z 707.31,A -85,B 0,C 180,E1 1275.312,E2 1275.312} C_VEL
LIN {X 0,Y 745.868,Z 707.31,A -85,B 0,C 180,E1 1280.836,E2 1280.836} C_VEL
LIN {X 0,Y 745.966,Z 707.31,A -85,B 0,C 180,E1 1286.639,E2 1286.639} C_VEL
LIN {X 0,Y 746.011,Z 707.31,A -85,B 0,C 180,E1 1291.877,E2 1291.877} C_VEL
LIN {X 0,Y 745.839,Z 707.31,A -85,B 0,C 180,E1 1296.099,E2 1296.099} C_VEL
LIN {X 0,Y 745.861,Z 707.31,A -85,B 0,C 180,E1 1300.55,E2 1300.55} C_VEL
LIN {X 0,Y 746.004,Z 707.31,A -85,B 0,C 180,E1 1305.311,E2 1305.311} C_VEL
LIN {X 0,Y 745.91,Z 707.31,A -85,B 0,C 180,E1 1310.964,E2 1310.964} C_VEL
LIN {X 0,Y 745.888,Z 707.31,A -85,B 0,C 180,E1 1315.328,E2 1315.328} C_VEL
LIN {X 0,Y 746.211,Z 708.049,A -85,B 0,C 180,E1 1319.734,E2 1319.734} C_VEL
LIN {X 0,Y 749.027,Z 721.889,A -85,B 0,C 180,E1 1320.01,E2 1320.01} C_VEL
LIN {X 0,Y 748.931,Z 789.558,A -85,B 0,C 180,E1 1320.874,E2 1320.874} C_VEL
LIN {X 0,Y 748.562,Z 838.058,A -85,B 0,C 180,E1 1322.08,E2 1322.08} C_VEL
LIN {X 0,Y 748.149,Z 884.93,A -85,B 0,C 180,E1 1323.853,E2 1323.853} C_VEL
LIN {X 0,Y 747.628,Z 927.895,A -85,B 0,C 180,E1 1326.084,E2 1326.084} C_VEL
LIN {X 0,Y 747.163,Z 967.678,A -85,B 0,C 180,E1 1328.805,E2 1328.805} C_VEL
LIN {X 0,Y 746.806,Z 1000.244,A -85,B 0,C 180,E1 1331.667,E2 1331.667} C_VEL
LIN {X 0,Y 746.516,Z 1029.535,A -85,B 0,C 180,E1 1334.999,E2 1334.999} C_VEL
LIN {X 0,Y 746.391,Z 1051.275,A -85,B 0,C 180,E1 1338.285,E2 1338.285} C_VEL
LIN {X 0,Y 746.341,Z 1066.859,A -85,B 0,C 180,E1 1341.534,E2 1341.534} C_VEL
LIN {X 0,Y 746.321,Z 1077.191,A -85,B 0,C 180,E1 1344.757,E2 1344.757} C_VEL
LIN {X 0,Y 746.338,Z 1082.219,A -85,B 0,C 180,E1 1347.672,E2 1347.672} C_VEL
LIN {X 0,Y 746.427,Z 1083.171,A -85,B 0,C 180,E1 1351.163,E2 1351.163} C_VEL
LIN {X 0,Y 746.322,Z 1078.46,A -85,B 0,C 180,E1 1354.658,E2 1354.658} C_VEL
LIN {X 0,Y 746.346,Z 1069.166,A -85,B 0,C 180,E1 1357.877,E2 1357.877} C_VEL
LIN {X 0,Y 746.493,Z 1052.975,A -85,B 0,C 180,E1 1361.415,E2 1361.415} C_VEL
LIN {X 0,Y 746.609,Z 1029.543,A -85,B 0,C 180,E1 1364.998,E2 1364.998} C_VEL
LIN {X 0,Y 746.859,Z 1000.255,A -85,B 0,C 180,E1 1368.33,E2 1368.33} C_VEL
LIN {X 0,Y 747.215,Z 966.286,A -85,B 0,C 180,E1 1371.304,E2 1371.304} C_VEL
LIN {X 0,Y 747.67,Z 927.917,A -85,B 0,C 180,E1 1373.913,E2 1373.913} C_VEL
LIN {X 0,Y 748.194,Z 884.961,A -85,B 0,C 180,E1 1376.144,E2 1376.144} C_VEL
LIN {X 0,Y 748.644,Z 841.607,A -85,B 0,C 180,E1 1377.799,E2 1377.799} C_VEL
LIN {X 0,Y 748.995,Z 799.12,A -85,B 0,C 180,E1 1378.922,E2 1378.922} C_VEL
LIN {X 0,Y 749.086,Z 754.307,A -85,B 0,C 180,E1 1379.637,E2 1379.637} C_VEL
LIN {X 0,Y 748.377,Z 716.318,A -85,B 0,C 180,E1 1380.079,E2 1380.079} C_VEL
LIN {X 0,Y 746.349,Z 707.31,A -85,B 0,C 180,E1 1380.295,E2 1380.295} C_VEL
LIN {X 0,Y 745.835,Z 707.31,A -85,B 0,C 180,E1 1386.101,E2 1386.101} C_VEL
LIN {X 0,Y 745.873,Z 707.31,A -85,B 0,C 180,E1 1390.552,E2 1390.552} C_VEL
LIN {X 0,Y 746.012,Z 707.31,A -85,B 0,C 180,E1 1395.313,E2 1395.313} C_VEL
LIN {X 0,Y 745.919,Z 707.31,A -85,B 0,C 180,E1 1400.969,E2 1400.969} C_VEL
LIN {X 0,Y 745.894,Z 707.31,A -85,B 0,C 180,E1 1406.405,E2 1406.405} C_VEL
LIN {X 0,Y 745.821,Z 707.31,A -85,B 0,C 180,E1 1410.89,E2 1410.89} C_VEL
LIN {X 0,Y 745.935,Z 707.31,A -85,B 0,C 180,E1 1414.749,E2 1414.749} C_VEL
LIN {X 0,Y 746.059,Z 707.31,A -85,B 0,C 180,E1 1419.802,E2 1419.802} C_VEL
LIN {X 0,Y 746.068,Z 707.31,A -85,B 0,C 180,E1 1425.895,E2 1425.895} C_VEL
LIN {X 0,Y 746.148,Z 707.31,A -85,B 0,C 180,E1 1430.652,E2 1430.652} C_VEL
LIN {X 0,Y 745.908,Z 707.31,A -85,B 0,C 180,E1 1434.551,E2 1434.551} C_VEL
LIN {X 0,Y 746.262,Z 707.31,A -85,B 0,C 180,E1 1438.839,E2 1438.839} C_VEL
LIN {X 0,Y 745.946,Z 707.31,A -85,B 0,C 180,E1 1445.48,E2 1445.48} C_VEL
LIN {X 0,Y 746.244,Z 707.31,A -85,B 0,C 180,E1 1450.533,E2 1450.533} C_VEL
LIN {X 0,Y 745.844,Z 707.31,A -85,B 0,C 180,E1 1455.317,E2 1455.317} C_VEL
LIN {X 0,Y 746.044,Z 707.31,A -85,B 0,C 180,E1 1460.875,E2 1460.875} C_VEL
LIN {X 0,Y 745.81,Z 707.31,A -85,B 0,C 180,E1 1465.26,E2 1465.26} C_VEL
LIN {X 0,Y 745.833,Z 707.31,A -85,B 0,C 180,E1 1470.53,E2 1470.53} C_VEL
LIN {X 0,Y 745.778,Z 707.31,A -85,B 0,C 180,E1 1476.107,E2 1476.107} C_VEL
LIN {X 0,Y 745.929,Z 707.31,A -85,B 0,C 180,E1 1480.551,E2 1480.551} C_VEL
LIN {X 0,Y 746.007,Z 707.31,A -85,B 0,C 180,E1 1485.316,E2 1485.316} C_VEL
LIN {X 0,Y 746.09,Z 707.31,A -85,B 0,C 180,E1 1490.977,E2 1490.977} C_VEL
LIN {X 0,Y 745.669,Z 707.31,A -85,B 0,C 180,E1 1495.318,E2 1495.318} C_VEL
LIN {X 0,Y 746.195,Z 707.31,A -85,B 0,C 180,E1 1498.002,E2 1498.002} C_VEL
LIN {X 0,Y 749.026,Z 716.059,A -85,B 0,C 180,E1 1498.226,E2 1498.226} C_VEL
LIN {X 0,Y 748.911,Z 765.18,A -85,B 0,C 180,E1 1498.946,E2 1498.946} C_VEL
LIN {X 0,Y 748.631,Z 809.987,A -85,B 0,C 180,E1 1500.101,E2 1500.101} C_VEL
LIN {X 0,Y 748.157,Z 853.676,A -85,B 0,C 180,E1 1501.754,E2 1501.754} C_VEL
LIN {X 0,Y 747.656,Z 895.833,A -85,B 0,C 180,E1 1503.921,E2 1503.921} C_VEL
LIN {X 0,Y 747.201,Z 933.827,A -85,B 0,C 180,E1 1506.467,E2 1506.467} C_VEL
LIN {X 0,Y 746.845,Z 967.913,A -85,B 0,C 180,E1 1509.399,E2 1509.399} C_VEL
LIN {X 0,Y 746.558,Z 996.446,A -85,B 0,C 180,E1 1512.564,E2 1512.564} C_VEL
LIN {X 0,Y 746.452,Z 1017.497,A -85,B 0,C 180,E1 1515.6,E2 1515.6} C_VEL
LIN {X 0,Y 746.431,Z 1034.417,A -85,B 0,C 180,E1 1518.88,E2 1518.88} C_VEL
LIN {X 0,Y 746.382,Z 1046.402,A -85,B 0,C 180,E1 1522.417,E2 1522.417} C_VEL
LIN {X 0,Y 746.297,Z 1051.936,A -85,B 0,C 180,E1 1525.342,E2 1525.342} C_VEL
LIN {X 0,Y 746.214,Z 1053.252,A -85,B 0,C 180,E1 1528.837,E2 1528.837} C_VEL
LIN {X 0,Y 746.274,Z 1049.047,A -85,B 0,C 180,E1 1532.328,E2 1532.328} C_VEL
LIN {X 0,Y 746.262,Z 1039.185,A -85,B 0,C 180,E1 1535.828,E2 1535.828} C_VEL
LIN {X 0,Y 746.28,Z 1024.636,A -85,B 0,C 180,E1 1539.055,E2 1539.055} C_VEL
LIN {X 0,Y 746.423,Z 1005.359,A -85,B 0,C 180,E1 1542.16,E2 1542.16} C_VEL
LIN {X 0,Y 746.695,Z 979.799,A -85,B 0,C 180,E1 1545.298,E2 1545.298} C_VEL
LIN {X 0,Y 747.02,Z 947.897,A -85,B 0,C 180,E1 1548.327,E2 1548.327} C_VEL
LIN {X 0,Y 747.482,Z 910.148,A -85,B 0,C 180,E1 1551.106,E2 1551.106} C_VEL
LIN {X 0,Y 748.042,Z 869.234,A -85,B 0,C 180,E1 1553.427,E2 1553.427} C_VEL
LIN {X 0,Y 748.546,Z 824.817,A -85,B 0,C 180,E1 1555.309,E2 1555.309} C_VEL
LIN {X 0,Y 748.869,Z 780.176,A -85,B 0,C 180,E1 1556.633,E2 1556.633} C_VEL
LIN {X 0,Y 749.188,Z 736.743,A -85,B 0,C 180,E1 1557.432,E2 1557.432} C_VEL
LIN {X 0,Y 748.27,Z 713.356,A -85,B 0,C 180,E1 1557.746,E2 1557.746} C_VEL
LIN {X 0,Y 746.195,Z 707.31,A -85,B 0,C 180,E1 1557.925,E2 1557.925} C_VEL
LIN {X 0,Y 745.752,Z 707.31,A -85,B 0,C 180,E1 1563.575,E2 1563.575} C_VEL
LIN {X 0,Y 745.965,Z 707.31,A -85,B 0,C 180,E1 1569.033,E2 1569.033} C_VEL
LIN {X 0,Y 746.081,Z 707.31,A -85,B 0,C 180,E1 1575.309,E2 1575.309} C_VEL
LIN {X 0,Y 745.933,Z 707.31,A -85,B 0,C 180,E1 1580.964,E2 1580.964} C_VEL
LIN {X 0,Y 745.887,Z 707.31,A -85,B 0,C 180,E1 1586.408,E2 1586.408} C_VEL
LIN {X 0,Y 745.812,Z 707.31,A -85,B 0,C 180,E1 1590.893,E2 1590.893} C_VEL
LIN {X 0,Y 745.975,Z 707.31,A -85,B 0,C 180,E1 1594.746,E2 1594.746} C_VEL
LIN {X 0,Y 746.101,Z 707.31,A -85,B 0,C 180,E1 1599.799,E2 1599.799} C_VEL
LIN {X 0,Y 746.171,Z 707.31,A -85,B 0,C 180,E1 1605.892,E2 1605.892} C_VEL
LIN {X 0,Y 746.123,Z 707.31,A -85,B 0,C 180,E1 1610.647,E2 1610.647} C_VEL
LIN {X 0,Y 746.289,Z 707.31,A -85,B 0,C 180,E1 1615.339,E2 1615.339} C_VEL
LIN {X 0,Y 745.8,Z 707.31,A -85,B 0,C 180,E1 1619.652,E2 1619.652} C_VEL
LIN {X 0,Y 742.083,Z 707.31,A -85,B 0,C 180,E1 1620.971,E2 1620.971} C_VEL
LIN {X 0,Y 737.912,Z 707.31,A -85,B 0,C 180,E1 1622.304,E2 1622.304} C_VEL
LIN {X 0,Y 738.364,Z 707.31,A -85,B 0,C 180,E1 1627.071,E2 1627.071} C_VEL
LIN {X 0,Y 738.079,Z 707.31,A -85,B 0,C 180,E1 1631.846,E2 1631.846} C_VEL
LIN {X 0,Y 737.989,Z 707.31,A -85,B 0,C 180,E1 1635.48,E2 1635.48} C_VEL
LIN {X 0,Y 738.096,Z 707.31,A -85,B 0,C 180,E1 1640.425,E2 1640.425} C_VEL
LIN {X 0,Y 738.035,Z 707.31,A -85,B 0,C 180,E1 1645.54,E2 1645.54} C_VEL
LIN {X 0,Y 738.178,Z 707.31,A -85,B 0,C 180,E1 1650.876,E2 1650.876} C_VEL
LIN {X 0,Y 738.032,Z 707.31,A -85,B 0,C 180,E1 1655.091,E2 1655.091} C_VEL
LIN {X 0,Y 737.978,Z 707.31,A -85,B 0,C 180,E1 1660.555,E2 1660.555} C_VEL
LIN {X 0,Y 737.966,Z 707.31,A -85,B 0,C 180,E1 1665.945,E2 1665.945} C_VEL
LIN {X 0,Y 737.961,Z 707.31,A -85,B 0,C 180,E1 1671.286,E2 1671.286} C_VEL
LIN {X 0,Y 737.857,Z 707.31,A -85,B 0,C 180,E1 1676.322,E2 1676.322} C_VEL
LIN {X 0,Y 738.102,Z 707.31,A -85,B 0,C 180,E1 1679.342,E2 1679.342} C_VEL
LIN {X 0,Y 742.131,Z 719.663,A -85,B 0,C 180,E1 1679.678,E2 1679.678} C_VEL
LIN {X 0,Y 742.015,Z 789.558,A -85,B 0,C 180,E1 1680.576,E2 1680.576} C_VEL
LIN {X 0,Y 741.505,Z 838.384,A -85,B 0,C 180,E1 1681.801,E2 1681.801} C_VEL
LIN {X 0,Y 740.902,Z 885.4,A -85,B 0,C 180,E1 1683.598,E2 1683.598} C_VEL
LIN {X 0,Y 740.192,Z 929.201,A -85,B 0,C 180,E1 1685.909,E2 1685.909} C_VEL
LIN {X 0,Y 739.609,Z 966.936,A -85,B 0,C 180,E1 1688.517,E2 1688.517} C_VEL
LIN {X 0,Y 739.102,Z 1000.245,A -85,B 0,C 180,E1 1691.47,E2 1691.47} C_VEL
LIN {X 0,Y 738.751,Z 1028.405,A -85,B 0,C 180,E1 1694.689,E2 1694.689} C_VEL
LIN {X 0,Y 738.541,Z 1051.277,A -85,B 0,C 180,E1 1698.159,E2 1698.159} C_VEL
LIN {X 0,Y 738.453,Z 1066.859,A -85,B 0,C 180,E1 1701.443,E2 1701.443} C_VEL
LIN {X 0,Y 738.412,Z 1077.444,A -85,B 0,C 180,E1 1704.799,E2 1704.799} C_VEL
LIN {X 0,Y 738.46,Z 1082.22,A -85,B 0,C 180,E1 1707.647,E2 1707.647} C_VEL
LIN {X 0,Y 738.524,Z 1083.17,A -85,B 0,C 180,E1 1711.175,E2 1711.175} C_VEL
LIN {X 0,Y 738.443,Z 1078.46,A -85,B 0,C 180,E1 1714.708,E2 1714.708} C_VEL
LIN {X 0,Y 738.458,Z 1069.166,A -85,B 0,C 180,E1 1717.962,E2 1717.962} C_VEL
LIN {X 0,Y 738.617,Z 1052.976,A -85,B 0,C 180,E1 1721.539,E2 1721.539} C_VEL
LIN {X 0,Y 738.802,Z 1029.767,A -85,B 0,C 180,E1 1725.129,E2 1725.129} C_VEL
LIN {X 0,Y 739.108,Z 1000.256,A -85,B 0,C 180,E1 1728.529,E2 1728.529} C_VEL
LIN {X 0,Y 739.627,Z 965.878,A -85,B 0,C 180,E1 1731.564,E2 1731.564} C_VEL
LIN {X 0,Y 740.283,Z 926.516,A -85,B 0,C 180,E1 1734.249,E2 1734.249} C_VEL
LIN {X 0,Y 740.981,Z 884.496,A -85,B 0,C 180,E1 1736.439,E2 1736.439} C_VEL
LIN {X 0,Y 741.618,Z 839.844,A -85,B 0,C 180,E1 1738.146,E2 1738.146} C_VEL
LIN {X 0,Y 742.071,Z 796.107,A -85,B 0,C 180,E1 1739.282,E2 1739.282} C_VEL
LIN {X 0,Y 742.225,Z 753.719,A -85,B 0,C 180,E1 1739.945,E2 1739.945} C_VEL
LIN {X 0,Y 741.663,Z 718.409,A -85,B 0,C 180,E1 1740.357,E2 1740.357} C_VEL
LIN {X 0,Y 738.364,Z 707.31,A -85,B 0,C 180,E1 1740.655,E2 1740.655} C_VEL
LIN {X 0,Y 738.032,Z 707.31,A -85,B 0,C 180,E1 1745.094,E2 1745.094} C_VEL
LIN {X 0,Y 737.988,Z 707.31,A -85,B 0,C 180,E1 1750.561,E2 1750.561} C_VEL
LIN {X 0,Y 737.971,Z 707.31,A -85,B 0,C 180,E1 1755.948,E2 1755.948} C_VEL
LIN {X 0,Y 737.974,Z 707.31,A -85,B 0,C 180,E1 1761.288,E2 1761.288} C_VEL
LIN {X 0,Y 737.991,Z 707.31,A -85,B 0,C 180,E1 1766.332,E2 1766.332} C_VEL
LIN {X 0,Y 737.977,Z 707.31,A -85,B 0,C 180,E1 1770.476,E2 1770.476} C_VEL
LIN {X 0,Y 738.032,Z 707.31,A -85,B 0,C 180,E1 1774.614,E2 1774.614} C_VEL
LIN {X 0,Y 738.03,Z 707.31,A -85,B 0,C 180,E1 1780.823,E2 1780.823} C_VEL
LIN {X 0,Y 738.127,Z 707.31,A -85,B 0,C 180,E1 1785.74,E2 1785.74} C_VEL
LIN {X 0,Y 738.252,Z 707.31,A -85,B 0,C 180,E1 1790.551,E2 1790.551} C_VEL
LIN {X 0,Y 738.153,Z 707.31,A -85,B 0,C 180,E1 1794.111,E2 1794.111} C_VEL
LIN {X 0,Y 738.356,Z 707.31,A -85,B 0,C 180,E1 1798.826,E2 1798.826} C_VEL
LIN {X 0,Y 738.381,Z 707.31,A -85,B 0,C 180,E1 1804.711,E2 1804.711} C_VEL
LIN {X 0,Y 738.294,Z 707.31,A -85,B 0,C 180,E1 1810.647,E2 1810.647} C_VEL
LIN {X 0,Y 737.897,Z 707.31,A -85,B 0,C 180,E1 1815.487,E2 1815.487} C_VEL
LIN {X 0,Y 738.203,Z 707.31,A -85,B 0,C 180,E1 1820.427,E2 1820.427} C_VEL
LIN {X 0,Y 737.905,Z 707.31,A -85,B 0,C 180,E1 1825.365,E2 1825.365} C_VEL
LIN {X 0,Y 737.858,Z 707.31,A -85,B 0,C 180,E1 1830.896,E2 1830.896} C_VEL
LIN {X 0,Y 737.952,Z 707.31,A -85,B 0,C 180,E1 1835.101,E2 1835.101} C_VEL
LIN {X 0,Y 738.042,Z 707.31,A -85,B 0,C 180,E1 1840.562,E2 1840.562} C_VEL
LIN {X 0,Y 737.976,Z 707.31,A -85,B 0,C 180,E1 1845.95,E2 1845.95} C_VEL
LIN {X 0,Y 738.171,Z 707.31,A -85,B 0,C 180,E1 1851.273,E2 1851.273} C_VEL
LIN {X 0,Y 737.786,Z 707.31,A -85,B 0,C 180,E1 1856.319,E2 1856.319} C_VEL
LIN {X 0,Y 738.147,Z 707.659,A -85,B 0,C 180,E1 1857.65,E2 1857.65} C_VEL
LIN {X 0,Y 742.184,Z 718.81,A -85,B 0,C 180,E1 1857.955,E2 1857.955} C_VEL
LIN {X 0,Y 741.965,Z 766.901,A -85,B 0,C 180,E1 1858.685,E2 1858.685} C_VEL
LIN {X 0,Y 741.553,Z 810.135,A -85,B 0,C 180,E1 1859.816,E2 1859.816} C_VEL
LIN {X 0,Y 740.902,Z 855.144,A -85,B 0,C 180,E1 1861.542,E2 1861.542} C_VEL
LIN {X 0,Y 740.246,Z 898.739,A -85,B 0,C 180,E1 1863.836,E2 1863.836} C_VEL
LIN {X 0,Y 739.626,Z 936.678,A -85,B 0,C 180,E1 1866.452,E2 1866.452} C_VEL
LIN {X 0,Y 739.133,Z 970.125,A -85,B 0,C 180,E1 1869.413,E2 1869.413} C_VEL
LIN {X 0,Y 738.763,Z 998.656,A -85,B 0,C 180,E1 1872.676,E2 1872.676} C_VEL
LIN {X 0,Y 738.621,Z 1022.647,A -85,B 0,C 180,E1 1876.353,E2 1876.353} C_VEL
LIN {X 0,Y 738.457,Z 1038.551,A -85,B 0,C 180,E1 1879.835,E2 1879.835} C_VEL
LIN {X 0,Y 738.412,Z 1049.016,A -85,B 0,C 180,E1 1883.52,E2 1883.52} C_VEL
LIN {X 0,Y 738.415,Z 1052.968,A -85,B 0,C 180,E1 1886.471,E2 1886.471} C_VEL
LIN {X 0,Y 738.475,Z 1052.484,A -85,B 0,C 180,E1 1890.001,E2 1890.001} C_VEL
LIN {X 0,Y 738.552,Z 1046.461,A -85,B 0,C 180,E1 1893.53,E2 1893.53} C_VEL
LIN {X 0,Y 738.568,Z 1034.662,A -85,B 0,C 180,E1 1897.072,E2 1897.072} C_VEL
LIN {X 0,Y 738.671,Z 1016.341,A -85,B 0,C 180,E1 1900.641,E2 1900.641} C_VEL
LIN {X 0,Y 738.887,Z 991.776,A -85,B 0,C 180,E1 1904.097,E2 1904.097} C_VEL
LIN {X 0,Y 739.266,Z 962.269,A -85,B 0,C 180,E1 1907.253,E2 1907.253} C_VEL
LIN {X 0,Y 739.731,Z 929.418,A -85,B 0,C 180,E1 1910.004,E2 1910.004} C_VEL
LIN {X 0,Y 740.294,Z 892.947,A -85,B 0,C 180,E1 1912.412,E2 1912.412} C_VEL
LIN {X 0,Y 741.012,Z 851.882,A -85,B 0,C 180,E1 1914.506,E2 1914.506} C_VEL
LIN {X 0,Y 741.514,Z 807.432,A -85,B 0,C 180,E1 1916.183,E2 1916.183} C_VEL
LIN {X 0,Y 742.1,Z 759.448,A -85,B 0,C 180,E1 1917.377,E2 1917.377} C_VEL
LIN {X 0,Y 741.381,Z 715.712,A -85,B 0,C 180,E1 1918.025,E2 1918.025} C_VEL
LIN {X 0,Y 738.245,Z 707.31,A -85,B 0,C 180,E1 1918.304,E2 1918.304} C_VEL
LIN {X 0,Y 737.86,Z 707.31,A -85,B 0,C 180,E1 1923.678,E2 1923.678} C_VEL
LIN {X 0,Y 738.008,Z 707.31,A -85,B 0,C 180,E1 1928.711,E2 1928.711} C_VEL
LIN {X 0,Y 738.018,Z 707.31,A -85,B 0,C 180,E1 1934.278,E2 1934.278} C_VEL
LIN {X 0,Y 738.043,Z 707.31,A -85,B 0,C 180,E1 1939.439,E2 1939.439} C_VEL
LIN {X 0,Y 738.033,Z 707.31,A -85,B 0,C 180,E1 1945.218,E2 1945.218} C_VEL
LIN {X 0,Y 737.944,Z 707.31,A -85,B 0,C 180,E1 1950.47,E2 1950.47} C_VEL
LIN {X 0,Y 738.059,Z 707.31,A -85,B 0,C 180,E1 1954.612,E2 1954.612} C_VEL
LIN {X 0,Y 738.029,Z 707.31,A -85,B 0,C 180,E1 1960.827,E2 1960.827} C_VEL
LIN {X 0,Y 738.396,Z 707.31,A -85,B 0,C 180,E1 1966.951,E2 1966.951} C_VEL
LIN {X 0,Y 738.261,Z 707.31,A -85,B 0,C 180,E1 1971.889,E2 1971.889} C_VEL
LIN {X 0,Y 737.959,Z 707.31,A -85,B 0,C 180,E1 1976.466,E2 1976.466} C_VEL
LIN {X 0,Y 738.386,Z 707.31,A -85,B 0,C 180,E1 1981.174,E2 1981.174} C_VEL
LIN {X 0,Y 737.912,Z 707.31,A -85,B 0,C 180,E1 1982.304,E2 1982.304} C_VEL
LIN {X 0,Y 733.767,Z 707.31,A -85,B 0,C 180,E1 1983.626,E2 1983.626} C_VEL
LIN {X 0,Y 729.954,Z 707.31,A -85,B 0,C 180,E1 1984.962,E2 1984.962} C_VEL
LIN {X 0,Y 730.25,Z 707.31,A -85,B 0,C 180,E1 1988.35,E2 1988.35} C_VEL
LIN {X 0,Y 730.139,Z 707.31,A -85,B 0,C 180,E1 1992.711,E2 1992.711} C_VEL
LIN {X 0,Y 729.846,Z 707.31,A -85,B 0,C 180,E1 1997.231,E2 1997.231} C_VEL
LIN {X 0,Y 730.049,Z 707.31,A -85,B 0,C 180,E1 2000.917,E2 2000.917} C_VEL
LIN {X 0,Y 730.113,Z 707.31,A -85,B 0,C 180,E1 2006.811,E2 2006.811} C_VEL
LIN {X 0,Y 730.141,Z 707.31,A -85,B 0,C 180,E1 2011.684,E2 2011.684} C_VEL
LIN {X 0,Y 730.009,Z 707.31,A -85,B 0,C 180,E1 2017.01,E2 2017.01} C_VEL
LIN {X 0,Y 729.895,Z 707.31,A -85,B 0,C 180,E1 2021.631,E2 2021.631} C_VEL
LIN {X 0,Y 729.917,Z 707.31,A -85,B 0,C 180,E1 2026.602,E2 2026.602} C_VEL
LIN {X 0,Y 730.037,Z 707.31,A -85,B 0,C 180,E1 2031.483,E2 2031.483} C_VEL
LIN {X 0,Y 729.973,Z 707.31,A -85,B 0,C 180,E1 2036.133,E2 2036.133} C_VEL
LIN {X 0,Y 730.146,Z 708.014,A -85,B 0,C 180,E1 2038.995,E2 2038.995} C_VEL
LIN {X 0,Y 735.275,Z 721.357,A -85,B 0,C 180,E1 2039.383,E2 2039.383} C_VEL
LIN {X 0,Y 735.145,Z 789.522,A -85,B 0,C 180,E1 2040.273,E2 2040.273} C_VEL
LIN {X 0,Y 734.477,Z 838.385,A -85,B 0,C 180,E1 2041.506,E2 2041.506} C_VEL
LIN {X 0,Y 733.659,Z 885.487,A -85,B 0,C 180,E1 2043.321,E2 2043.321} C_VEL
LIN {X 0,Y 732.784,Z 928.969,A -85,B 0,C 180,E1 2045.635,E2 2045.635} C_VEL
LIN {X 0,Y 732.013,Z 968.185,A -85,B 0,C 180,E1 2048.386,E2 2048.386} C_VEL
LIN {X 0,Y 731.368,Z 1001.72,A -85,B 0,C 180,E1 2051.423,E2 2051.423} C_VEL
LIN {X 0,Y 730.922,Z 1029.819,A -85,B 0,C 180,E1 2054.711,E2 2054.711} C_VEL
LIN {X 0,Y 730.698,Z 1051.277,A -85,B 0,C 180,E1 2058.03,E2 2058.03} C_VEL
LIN {X 0,Y 730.584,Z 1066.859,A -85,B 0,C 180,E1 2061.35,E2 2061.35} C_VEL
LIN {X 0,Y 730.54,Z 1077.203,A -85,B 0,C 180,E1 2064.648,E2 2064.648} C_VEL
LIN {X 0,Y 730.556,Z 1082.22,A -85,B 0,C 180,E1 2067.622,E2 2067.622} C_VEL
LIN {X 0,Y 730.621,Z 1083.17,A -85,B 0,C 180,E1 2071.188,E2 2071.188} C_VEL
LIN {X 0,Y 730.539,Z 1078.46,A -85,B 0,C 180,E1 2074.759,E2 2074.759} C_VEL
LIN {X 0,Y 730.548,Z 1069.166,A -85,B 0,C 180,E1 2078.048,E2 2078.048} C_VEL
LIN {X 0,Y 730.731,Z 1052.977,A -85,B 0,C 180,E1 2081.665,E2 2081.665} C_VEL
LIN {X 0,Y 730.984,Z 1029.816,A -85,B 0,C 180,E1 2085.288,E2 2085.288} C_VEL
LIN {X 0,Y 731.397,Z 1000.257,A -85,B 0,C 180,E1 2088.732,E2 2088.732} C_VEL
LIN {X 0,Y 732.048,Z 965.994,A -85,B 0,C 180,E1 2091.79,E2 2091.79} C_VEL
LIN {X 0,Y 732.855,Z 927.923,A -85,B 0,C 180,E1 2094.428,E2 2094.428} C_VEL
LIN {X 0,Y 733.752,Z 885.545,A -85,B 0,C 180,E1 2096.672,E2 2096.672} C_VEL
LIN {X 0,Y 734.528,Z 842.068,A -85,B 0,C 180,E1 2098.365,E2 2098.365} C_VEL
LIN {X 0,Y 735.131,Z 800.413,A -85,B 0,C 180,E1 2099.493,E2 2099.493} C_VEL
LIN {X 0,Y 735.372,Z 756.884,A -85,B 0,C 180,E1 2100.217,E2 2100.217} C_VEL
LIN {X 0,Y 734.632,Z 719.113,A -85,B 0,C 180,E1 2100.671,E2 2100.671} C_VEL
LIN {X 0,Y 730.323,Z 707.31,A -85,B 0,C 180,E1 2101.073,E2 2101.073} C_VEL
LIN {X 0,Y 730.013,Z 707.31,A -85,B 0,C 180,E1 2105.95,E2 2105.95} C_VEL
LIN {X 0,Y 730.114,Z 707.31,A -85,B 0,C 180,E1 2110.047,E2 2110.047} C_VEL
LIN {X 0,Y 730.092,Z 707.31,A -85,B 0,C 180,E1 2115.117,E2 2115.117} C_VEL
LIN {X 0,Y 730.121,Z 707.31,A -85,B 0,C 180,E1 2120.169,E2 2120.169} C_VEL
LIN {X 0,Y 730.098,Z 707.31,A -85,B 0,C 180,E1 2125.919,E2 2125.919} C_VEL
LIN {X 0,Y 730.036,Z 707.31,A -85,B 0,C 180,E1 2130.671,E2 2130.671} C_VEL
LIN {X 0,Y 729.95,Z 707.31,A -85,B 0,C 180,E1 2135.47,E2 2135.47} C_VEL
LIN {X 0,Y 730.117,Z 707.31,A -85,B 0,C 180,E1 2140.607,E2 2140.607} C_VEL
LIN {X 0,Y 730.198,Z 707.31,A -85,B 0,C 180,E1 2145.582,E2 2145.582} C_VEL
LIN {X 0,Y 730.359,Z 707.31,A -85,B 0,C 180,E1 2150.448,E2 2150.448} C_VEL
LIN {X 0,Y 730.257,Z 707.31,A -85,B 0,C 180,E1 2154.047,E2 2154.047} C_VEL
LIN {X 0,Y 730.444,Z 707.31,A -85,B 0,C 180,E1 2158.813,E2 2158.813} C_VEL
LIN {X 0,Y 730.286,Z 707.31,A -85,B 0,C 180,E1 2165.11,E2 2165.11} C_VEL
LIN {X 0,Y 730.349,Z 707.31,A -85,B 0,C 180,E1 2170.765,E2 2170.765} C_VEL
LIN {X 0,Y 729.957,Z 707.31,A -85,B 0,C 180,E1 2175.659,E2 2175.659} C_VEL
LIN {X 0,Y 730.213,Z 707.31,A -85,B 0,C 180,E1 2180.954,E2 2180.954} C_VEL
LIN {X 0,Y 730.185,Z 707.31,A -85,B 0,C 180,E1 2184.526,E2 2184.526} C_VEL
LIN {X 0,Y 729.992,Z 707.31,A -85,B 0,C 180,E1 2189.884,E2 2189.884} C_VEL
LIN {X 0,Y 729.968,Z 707.31,A -85,B 0,C 180,E1 2195.542,E2 2195.542} C_VEL
LIN {X 0,Y 730.146,Z 707.31,A -85,B 0,C 180,E1 2200.048,E2 2200.048} C_VEL
LIN {X 0,Y 730.1,Z 707.31,A -85,B 0,C 180,E1 2205.114,E2 2205.114} C_VEL
LIN {X 0,Y 730.265,Z 707.31,A -85,B 0,C 180,E1 2211.499,E2 2211.499} C_VEL
LIN {X 0,Y 730.104,Z 707.31,A -85,B 0,C 180,E1 2217.266,E2 2217.266} C_VEL
LIN {X 0,Y 735.382,Z 722.55,A -85,B 0,C 180,E1 2217.689,E2 2217.689} C_VEL
LIN {X 0,Y 735.017,Z 770.462,A -85,B 0,C 180,E1 2218.458,E2 2218.458} C_VEL
LIN {X 0,Y 734.431,Z 813.122,A -85,B 0,C 180,E1 2219.622,E2 2219.622} C_VEL
LIN {X 0,Y 733.616,Z 857.276,A -85,B 0,C 180,E1 2221.361,E2 2221.361} C_VEL
LIN {X 0,Y 732.812,Z 899.155,A -85,B 0,C 180,E1 2223.603,E2 2223.603} C_VEL
LIN {X 0,Y 732.007,Z 936.761,A -85,B 0,C 180,E1 2226.223,E2 2226.223} C_VEL
LIN {X 0,Y 731.38,Z 970.369,A -85,B 0,C 180,E1 2229.235,E2 2229.235} C_VEL
LIN {X 0,Y 730.966,Z 999.269,A -85,B 0,C 180,E1 2232.59,E2 2232.59} C_VEL
LIN {X 0,Y 730.785,Z 1022.521,A -85,B 0,C 180,E1 2236.204,E2 2236.204} C_VEL
LIN {X 0,Y 730.534,Z 1039.483,A -85,B 0,C 180,E1 2239.989,E2 2239.989} C_VEL
LIN {X 0,Y 730.532,Z 1048.971,A -85,B 0,C 180,E1 2243.449,E2 2243.449} C_VEL
LIN {X 0,Y 730.511,Z 1052.949,A -85,B 0,C 180,E1 2246.433,E2 2246.433} C_VEL
LIN {X 0,Y 730.574,Z 1052.503,A -85,B 0,C 180,E1 2250.001,E2 2250.001} C_VEL
LIN {X 0,Y 730.644,Z 1046.52,A -85,B 0,C 180,E1 2253.568,E2 2253.568} C_VEL
LIN {X 0,Y 730.691,Z 1034.758,A -85,B 0,C 180,E1 2257.149,E2 2257.149} C_VEL
LIN {X 0,Y 730.802,Z 1016.475,A -85,B 0,C 180,E1 2260.756,E2 2260.756} C_VEL
LIN {X 0,Y 731.087,Z 991.962,A -85,B 0,C 180,E1 2264.25,E2 2264.25} C_VEL
LIN {X 0,Y 731.56,Z 962.945,A -85,B 0,C 180,E1 2267.398,E2 2267.398} C_VEL
LIN {X 0,Y 732.184,Z 929.046,A -85,B 0,C 180,E1 2270.272,E2 2270.272} C_VEL
LIN {X 0,Y 732.932,Z 892.163,A -85,B 0,C 180,E1 2272.721,E2 2272.721} C_VEL
LIN {X 0,Y 733.81,Z 851.952,A -85,B 0,C 180,E1 2274.785,E2 2274.785} C_VEL
LIN {X 0,Y 734.512,Z 807.058,A -85,B 0,C 180,E1 2276.488,E2 2276.488} C_VEL
LIN {X 0,Y 735.184,Z 760.163,A -85,B 0,C 180,E1 2277.667,E2 2277.667} C_VEL
LIN {X 0,Y 734.702,Z 718.625,A -85,B 0,C 180,E1 2278.295,E2 2278.295} C_VEL
LIN {X 0,Y 730.318,Z 707.31,A -85,B 0,C 180,E1 2278.676,E2 2278.676} C_VEL
LIN {X 0,Y 729.998,Z 707.31,A -85,B 0,C 180,E1 2284.09,E2 2284.09} C_VEL
LIN {X 0,Y 730.17,Z 707.31,A -85,B 0,C 180,E1 2289.832,E2 2289.832} C_VEL
LIN {X 0,Y 730.119,Z 707.31,A -85,B 0,C 180,E1 2295.113,E2 2295.113} C_VEL
LIN {X 0,Y 730.158,Z 707.31,A -85,B 0,C 180,E1 2300.168,E2 2300.168} C_VEL
LIN {X 0,Y 730.096,Z 707.31,A -85,B 0,C 180,E1 2305.913,E2 2305.913} C_VEL
LIN {X 0,Y 730.012,Z 707.31,A -85,B 0,C 180,E1 2310.676,E2 2310.676} C_VEL
LIN {X 0,Y 729.982,Z 707.31,A -85,B 0,C 180,E1 2315.467,E2 2315.467} C_VEL
LIN {X 0,Y 730.12,Z 707.31,A -85,B 0,C 180,E1 2320.602,E2 2320.602} C_VEL
LIN {X 0,Y 730.479,Z 707.31,A -85,B 0,C 180,E1 2327.171,E2 2327.171} C_VEL
LIN {X 0,Y 730.232,Z 707.31,A -85,B 0,C 180,E1 2332.845,E2 2332.845} C_VEL
LIN {X 0,Y 730.068,Z 707.31,A -85,B 0,C 180,E1 2336.428,E2 2336.428} C_VEL
LIN {X 0,Y 730.473,Z 707.31,A -85,B 0,C 180,E1 2341.187,E2 2341.187} C_VEL
LIN {X 0,Y 729.954,Z 707.31,A -85,B 0,C 180,E1 2344.962,E2 2344.962} C_VEL
LIN {X 0,Y 726.338,Z 707.31,A -85,B 0,C 180,E1 2346.306,E2 2346.306} C_VEL
LIN {X 0,Y 722.433,Z 707.31,A -85,B 0,C 180,E1 2347.663,E2 2347.663} C_VEL
LIN {X 0,Y 722.251,Z 707.31,A -85,B 0,C 180,E1 2352.109,E2 2352.109} C_VEL
LIN {X 0,Y 721.958,Z 707.31,A -85,B 0,C 180,E1 2357.087,E2 2357.087} C_VEL
LIN {X 0,Y 722.163,Z 707.31,A -85,B 0,C 180,E1 2360.897,E2 2360.897} C_VEL
LIN {X 0,Y 722.192,Z 707.31,A -85,B 0,C 180,E1 2366.143,E2 2366.143} C_VEL
LIN {X 0,Y 722.277,Z 707.31,A -85,B 0,C 180,E1 2371.633,E2 2371.633} C_VEL
LIN {X 0,Y 722.129,Z 707.31,A -85,B 0,C 180,E1 2377.113,E2 2377.113} C_VEL
LIN {X 0,Y 721.954,Z 707.31,A -85,B 0,C 180,E1 2382.194,E2 2382.194} C_VEL
LIN {X 0,Y 722.033,Z 707.31,A -85,B 0,C 180,E1 2386.163,E2 2386.163} C_VEL
LIN {X 0,Y 722.123,Z 707.31,A -85,B 0,C 180,E1 2390.982,E2 2390.982} C_VEL
LIN {X 0,Y 722.044,Z 707.31,A -85,B 0,C 180,E1 2395.481,E2 2395.481} C_VEL
LIN {X 0,Y 722.097,Z 707.31,A -85,B 0,C 180,E1 2398.591,E2 2398.591} C_VEL
LIN {X 0,Y 728.521,Z 723.441,A -85,B 0,C 180,E1 2399.092,E2 2399.092} C_VEL
LIN {X 0,Y 728.287,Z 789.521,A -85,B 0,C 180,E1 2399.965,E2 2399.965} C_VEL
LIN {X 0,Y 727.499,Z 837.946,A -85,B 0,C 180,E1 2401.194,E2 2401.194} C_VEL
LIN {X 0,Y 726.453,Z 884.939,A -85,B 0,C 180,E1 2403.01,E2 2403.01} C_VEL
LIN {X 0,Y 725.379,Z 928.966,A -85,B 0,C 180,E1 2405.37,E2 2405.37} C_VEL
LIN {X 0,Y 724.475,Z 966.729,A -85,B 0,C 180,E1 2408.028,E2 2408.028} C_VEL
LIN {X 0,Y 723.706,Z 1000.246,A -85,B 0,C 180,E1 2411.06,E2 2411.06} C_VEL
LIN {X 0,Y 723.206,Z 1029.027,A -85,B 0,C 180,E1 2414.433,E2 2414.433} C_VEL
LIN {X 0,Y 722.858,Z 1051.276,A -85,B 0,C 180,E1 2417.898,E2 2417.898} C_VEL
LIN {X 0,Y 722.713,Z 1066.859,A -85,B 0,C 180,E1 2421.255,E2 2421.255} C_VEL
LIN {X 0,Y 722.65,Z 1077.203,A -85,B 0,C 180,E1 2424.589,E2 2424.589} C_VEL
LIN {X 0,Y 722.678,Z 1082.219,A -85,B 0,C 180,E1 2427.596,E2 2427.596} C_VEL
LIN {X 0,Y 722.719,Z 1083.17,A -85,B 0,C 180,E1 2431.201,E2 2431.201} C_VEL
LIN {X 0,Y 722.637,Z 1078.461,A -85,B 0,C 180,E1 2434.811,E2 2434.811} C_VEL
LIN {X 0,Y 722.641,Z 1069.166,A -85,B 0,C 180,E1 2438.137,E2 2438.137} C_VEL
LIN {X 0,Y 722.862,Z 1052.978,A -85,B 0,C 180,E1 2441.794,E2 2441.794} C_VEL
LIN {X 0,Y 723.171,Z 1029.89,A -85,B 0,C 180,E1 2445.447,E2 2445.447} C_VEL
LIN {X 0,Y 723.663,Z 1001.733,A -85,B 0,C 180,E1 2448.781,E2 2448.781} C_VEL
LIN {X 0,Y 724.422,Z 968.122,A -85,B 0,C 180,E1 2451.857,E2 2451.857} C_VEL
LIN {X 0,Y 725.41,Z 929.555,A -85,B 0,C 180,E1 2454.591,E2 2454.591} C_VEL
LIN {X 0,Y 726.454,Z 888.343,A -85,B 0,C 180,E1 2456.824,E2 2456.824} C_VEL
LIN {X 0,Y 727.4,Z 846.57,A -85,B 0,C 180,E1 2458.511,E2 2458.511} C_VEL
LIN {X 0,Y 728.174,Z 804.472,A -85,B 0,C 180,E1 2459.715,E2 2459.715} C_VEL
LIN {X 0,Y 728.549,Z 758.671,A -85,B 0,C 180,E1 2460.506,E2 2460.506} C_VEL
LIN {X 0,Y 727.758,Z 720.23,A -85,B 0,C 180,E1 2460.98,E2 2460.98} C_VEL
LIN {X 0,Y 722.36,Z 707.31,A -85,B 0,C 180,E1 2461.402,E2 2461.402} C_VEL
LIN {X 0,Y 722.128,Z 707.31,A -85,B 0,C 180,E1 2467.118,E2 2467.118} C_VEL
LIN {X 0,Y 722.014,Z 707.31,A -85,B 0,C 180,E1 2472.192,E2 2472.192} C_VEL
LIN {X 0,Y 722.035,Z 707.31,A -85,B 0,C 180,E1 2476.167,E2 2476.167} C_VEL
LIN {X 0,Y 722.134,Z 707.31,A -85,B 0,C 180,E1 2480.986,E2 2480.986} C_VEL
LIN {X 0,Y 722.134,Z 707.31,A -85,B 0,C 180,E1 2485.49,E2 2485.49} C_VEL
LIN {X 0,Y 722.205,Z 707.31,A -85,B 0,C 180,E1 2489.765,E2 2489.765} C_VEL
LIN {X 0,Y 722.049,Z 707.31,A -85,B 0,C 180,E1 2495.184,E2 2495.184} C_VEL
LIN {X 0,Y 722.193,Z 707.31,A -85,B 0,C 180,E1 2500.776,E2 2500.776} C_VEL
LIN {X 0,Y 722.248,Z 707.31,A -85,B 0,C 180,E1 2506.658,E2 2506.658} C_VEL
LIN {X 0,Y 722.469,Z 707.31,A -85,B 0,C 180,E1 2510.342,E2 2510.342} C_VEL
LIN {X 0,Y 722.361,Z 707.31,A -85,B 0,C 180,E1 2513.981,E2 2513.981} C_VEL
LIN {X 0,Y 722.542,Z 707.31,A -85,B 0,C 180,E1 2518.8,E2 2518.8} C_VEL
LIN {X 0,Y 722.527,Z 707.31,A -85,B 0,C 180,E1 2524.815,E2 2524.815} C_VEL
LIN {X 0,Y 722.406,Z 707.31,A -85,B 0,C 180,E1 2530.884,E2 2530.884} C_VEL
LIN {X 0,Y 722.019,Z 707.31,A -85,B 0,C 180,E1 2535.836,E2 2535.836} C_VEL
LIN {X 0,Y 722.349,Z 707.31,A -85,B 0,C 180,E1 2540.896,E2 2540.896} C_VEL
LIN {X 0,Y 722.051,Z 707.31,A -85,B 0,C 180,E1 2545.518,E2 2545.518} C_VEL
LIN {X 0,Y 721.978,Z 707.31,A -85,B 0,C 180,E1 2550.62,E2 2550.62} C_VEL
LIN {X 0,Y 722.064,Z 707.31,A -85,B 0,C 180,E1 2555.992,E2 2555.992} C_VEL
LIN {X 0,Y 722.108,Z 707.31,A -85,B 0,C 180,E1 2560.933,E2 2560.933} C_VEL
LIN {X 0,Y 722.033,Z 707.31,A -85,B 0,C 180,E1 2566.164,E2 2566.164} C_VEL
LIN {X 0,Y 722.297,Z 707.31,A -85,B 0,C 180,E1 2570.994,E2 2570.994} C_VEL
LIN {X 0,Y 722.023,Z 707.31,A -85,B 0,C 180,E1 2576.355,E2 2576.355} C_VEL
LIN {X 0,Y 722.127,Z 707.879,A -85,B 0,C 180,E1 2576.907,E2 2576.907} C_VEL
LIN {X 0,Y 728.573,Z 724.603,A -85,B 0,C 180,E1 2577.4,E2 2577.4} C_VEL
LIN {X 0,Y 728.106,Z 773.183,A -85,B 0,C 180,E1 2578.209,E2 2578.209} C_VEL
LIN {X 0,Y 727.326,Z 816.246,A -85,B 0,C 180,E1 2579.429,E2 2579.429} C_VEL
LIN {X 0,Y 726.359,Z 858.92,A -85,B 0,C 180,E1 2581.155,E2 2581.155} C_VEL
LIN {X 0,Y 725.407,Z 900.044,A -85,B 0,C 180,E1 2583.396,E2 2583.396} C_VEL
LIN {X 0,Y 724.409,Z 937.179,A -85,B 0,C 180,E1 2586.018,E2 2586.018} C_VEL
LIN {X 0,Y 723.654,Z 971.477,A -85,B 0,C 180,E1 2589.146,E2 2589.146} C_VEL
LIN {X 0,Y 723.156,Z 999.544,A -85,B 0,C 180,E1 2592.458,E2 2592.458} C_VEL
LIN {X 0,Y 722.917,Z 1022.39,A -85,B 0,C 180,E1 2596.051,E2 2596.051} C_VEL
LIN {X 0,Y 722.683,Z 1038.846,A -85,B 0,C 180,E1 2599.734,E2 2599.734} C_VEL
LIN {X 0,Y 722.661,Z 1048.927,A -85,B 0,C 180,E1 2603.378,E2 2603.378} C_VEL
LIN {X 0,Y 722.619,Z 1052.931,A -85,B 0,C 180,E1 2606.394,E2 2606.394} C_VEL
LIN {X 0,Y 722.703,Z 1052.522,A -85,B 0,C 180,E1 2610.001,E2 2610.001} C_VEL
LIN {X 0,Y 722.742,Z 1046.578,A -85,B 0,C 180,E1 2613.607,E2 2613.607} C_VEL
LIN {X 0,Y 722.785,Z 1034.852,A -85,B 0,C 180,E1 2617.227,E2 2617.227} C_VEL
LIN {X 0,Y 722.947,Z 1016.608,A -85,B 0,C 180,E1 2620.875,E2 2620.875} C_VEL
LIN {X 0,Y 723.271,Z 993.353,A -85,B 0,C 180,E1 2624.253,E2 2624.253} C_VEL
LIN {X 0,Y 723.832,Z 965.247,A -85,B 0,C 180,E1 2627.387,E2 2627.387} C_VEL
LIN {X 0,Y 724.61,Z 932.204,A -85,B 0,C 180,E1 2630.273,E2 2630.273} C_VEL
LIN {X 0,Y 725.49,Z 895.841,A -85,B 0,C 180,E1 2632.772,E2 2632.772} C_VEL
LIN {X 0,Y 726.588,Z 853.039,A -85,B 0,C 180,E1 2635.025,E2 2635.025} C_VEL
LIN {X 0,Y 727.505,Z 807.549,A -85,B 0,C 180,E1 2636.773,E2 2636.773} C_VEL
LIN {X 0,Y 728.302,Z 760.645,A -85,B 0,C 180,E1 2637.966,E2 2637.966} C_VEL
LIN {X 0,Y 727.903,Z 720.857,A -85,B 0,C 180,E1 2638.584,E2 2638.584} C_VEL
LIN {X 0,Y 722.376,Z 707.31,A -85,B 0,C 180,E1 2639.021,E2 2639.021} C_VEL
LIN {X 0,Y 722.058,Z 707.31,A -85,B 0,C 180,E1 2645.062,E2 2645.062} C_VEL
LIN {X 0,Y 722.171,Z 707.31,A -85,B 0,C 180,E1 2649.065,E2 2649.065} C_VEL
LIN {X 0,Y 722.123,Z 707.31,A -85,B 0,C 180,E1 2654.477,E2 2654.477} C_VEL
LIN {X 0,Y 722.129,Z 707.31,A -85,B 0,C 180,E1 2659.415,E2 2659.415} C_VEL
LIN {X 0,Y 722.133,Z 707.31,A -85,B 0,C 180,E1 2664.928,E2 2664.928} C_VEL
LIN {X 0,Y 722.191,Z 707.31,A -85,B 0,C 180,E1 2669.759,E2 2669.759} C_VEL
LIN {X 0,Y 722.079,Z 707.31,A -85,B 0,C 180,E1 2675.18,E2 2675.18} C_VEL
LIN {X 0,Y 722.171,Z 707.31,A -85,B 0,C 180,E1 2680.784,E2 2680.784} C_VEL
LIN {X 0,Y 722.529,Z 707.31,A -85,B 0,C 180,E1 2686.659,E2 2686.659} C_VEL
LIN {X 0,Y 722.417,Z 707.31,A -85,B 0,C 180,E1 2691.869,E2 2691.869} C_VEL
LIN {X 0,Y 722.206,Z 707.31,A -85,B 0,C 180,E1 2696.389,E2 2696.389} C_VEL
LIN {X 0,Y 722.57,Z 707.31,A -85,B 0,C 180,E1 2701.2,E2 2701.2} C_VEL
LIN {X 0,Y 722.433,Z 707.31,A -85,B 0,C 180,E1 2707.663,E2 2707.663} C_VEL
LIN {X 0,Y 718.421,Z 707.31,A -85,B 0,C 180,E1 2709.014,E2 2709.014} C_VEL
LIN {X 0,Y 714.543,Z 707.31,A -85,B 0,C 180,E1 2710.38,E2 2710.38} C_VEL
LIN {X 0,Y 714.343,Z 707.31,A -85,B 0,C 180,E1 2714.745,E2 2714.745} C_VEL
LIN {X 0,Y 714.287,Z 707.31,A -85,B 0,C 180,E1 2719.841,E2 2719.841} C_VEL
LIN {X 0,Y 714.195,Z 707.31,A -85,B 0,C 180,E1 2725.108,E2 2725.108} C_VEL
LIN {X 0,Y 714.339,Z 707.31,A -85,B 0,C 180,E1 2730.603,E2 2730.603} C_VEL
LIN {X 0,Y 714.212,Z 707.31,A -85,B 0,C 180,E1 2736.265,E2 2736.265} C_VEL
LIN {X 0,Y 714.087,Z 707.31,A -85,B 0,C 180,E1 2741.134,E2 2741.134} C_VEL
LIN {X 0,Y 714.131,Z 707.31,A -85,B 0,C 180,E1 2746.173,E2 2746.173} C_VEL
LIN {X 0,Y 714.164,Z 707.31,A -85,B 0,C 180,E1 2751.726,E2 2751.726} C_VEL
LIN {X 0,Y 714.048,Z 707.31,A -85,B 0,C 180,E1 2756.51,E2 2756.51} C_VEL
LIN {X 0,Y 714.108,Z 707.31,A -85,B 0,C 180,E1 2758.205,E2 2758.205} C_VEL
LIN {X 0,Y 721.796,Z 726.496,A -85,B 0,C 180,E1 2758.807,E2 2758.807} C_VEL
LIN {X 0,Y 721.438,Z 789.569,A -85,B 0,C 180,E1 2759.651,E2 2759.651} C_VEL
LIN {X 0,Y 720.505,Z 837.949,A -85,B 0,C 180,E1 2760.887,E2 2760.887} C_VEL
LIN {X 0,Y 719.299,Z 883.244,A -85,B 0,C 180,E1 2762.642,E2 2762.642} C_VEL
LIN {X 0,Y 718.058,Z 926.529,A -85,B 0,C 180,E1 2764.95,E2 2764.95} C_VEL
LIN {X 0,Y 716.993,Z 964.849,A -85,B 0,C 180,E1 2767.639,E2 2767.639} C_VEL
LIN {X 0,Y 716.039,Z 999.148,A -85,B 0,C 180,E1 2770.738,E2 2770.738} C_VEL
LIN {X 0,Y 715.428,Z 1029.025,A -85,B 0,C 180,E1 2774.259,E2 2774.259} C_VEL
LIN {X 0,Y 715.02,Z 1051.275,A -85,B 0,C 180,E1 2777.763,E2 2777.763} C_VEL
LIN {X 0,Y 714.848,Z 1066.86,A -85,B 0,C 180,E1 2781.158,E2 2781.158} C_VEL
LIN {X 0,Y 714.772,Z 1077.192,A -85,B 0,C 180,E1 2784.525,E2 2784.525} C_VEL
LIN {X 0,Y 714.773,Z 1082.219,A -85,B 0,C 180,E1 2787.569,E2 2787.569} C_VEL
LIN {X 0,Y 714.817,Z 1083.17,A -85,B 0,C 180,E1 2791.214,E2 2791.214} C_VEL
LIN {X 0,Y 714.738,Z 1078.461,A -85,B 0,C 180,E1 2794.864,E2 2794.864} C_VEL
LIN {X 0,Y 714.752,Z 1069.166,A -85,B 0,C 180,E1 2798.227,E2 2798.227} C_VEL
LIN {X 0,Y 714.991,Z 1052.979,A -85,B 0,C 180,E1 2801.925,E2 2801.925} C_VEL
LIN {X 0,Y 715.344,Z 1030.627,A -85,B 0,C 180,E1 2805.515,E2 2805.515} C_VEL
LIN {X 0,Y 715.915,Z 1003.427,A -85,B 0,C 180,E1 2808.808,E2 2808.808} C_VEL
LIN {X 0,Y 716.753,Z 972.184,A -85,B 0,C 180,E1 2811.758,E2 2811.758} C_VEL
LIN {X 0,Y 717.825,Z 936.656,A -85,B 0,C 180,E1 2814.399,E2 2814.399} C_VEL
LIN {X 0,Y 719.024,Z 896.735,A -85,B 0,C 180,E1 2816.704,E2 2816.704} C_VEL
LIN {X 0,Y 720.195,Z 853.671,A -85,B 0,C 180,E1 2818.57,E2 2818.57} C_VEL
LIN {X 0,Y 721.18,Z 808.24,A -85,B 0,C 180,E1 2819.939,E2 2819.939} C_VEL
LIN {X 0,Y 721.667,Z 763.758,A -85,B 0,C 180,E1 2820.76,E2 2820.76} C_VEL
LIN {X 0,Y 721.247,Z 723.393,A -85,B 0,C 180,E1 2821.255,E2 2821.255} C_VEL
LIN {X 0,Y 714.4,Z 707.31,A -85,B 0,C 180,E1 2821.802,E2 2821.802} C_VEL
LIN {X 0,Y 714.201,Z 707.31,A -85,B 0,C 180,E1 2826.448,E2 2826.448} C_VEL
LIN {X 0,Y 714.14,Z 707.31,A -85,B 0,C 180,E1 2831.133,E2 2831.133} C_VEL
LIN {X 0,Y 714.133,Z 707.31,A -85,B 0,C 180,E1 2836.176,E2 2836.176} C_VEL
LIN {X 0,Y 714.179,Z 707.31,A -85,B 0,C 180,E1 2841.728,E2 2841.728} C_VEL
LIN {X 0,Y 714.202,Z 707.31,A -85,B 0,C 180,E1 2846.521,E2 2846.521} C_VEL
LIN {X 0,Y 714.161,Z 707.31,A -85,B 0,C 180,E1 2850.791,E2 2850.791} C_VEL
LIN {X 0,Y 714.049,Z 707.31,A -85,B 0,C 180,E1 2855.862,E2 2855.862} C_VEL
LIN {X 0,Y 714.279,Z 707.31,A -85,B 0,C 180,E1 2860.159,E2 2860.159} C_VEL
LIN {X 0,Y 714.334,Z 707.31,A -85,B 0,C 180,E1 2865.254,E2 2865.254} C_VEL
LIN {X 0,Y 714.561,Z 707.31,A -85,B 0,C 180,E1 2870.234,E2 2870.234} C_VEL
LIN {X 0,Y 714.466,Z 707.31,A -85,B 0,C 180,E1 2873.915,E2 2873.915} C_VEL
LIN {X 0,Y 714.629,Z 707.31,A -85,B 0,C 180,E1 2878.787,E2 2878.787} C_VEL
LIN {X 0,Y 714.6,Z 707.31,A -85,B 0,C 180,E1 2884.868,E2 2884.868} C_VEL
LIN {X 0,Y 714.467,Z 707.31,A -85,B 0,C 180,E1 2891.007,E2 2891.007} C_VEL
LIN {X 0,Y 714.085,Z 707.31,A -85,B 0,C 180,E1 2896.017,E2 2896.017} C_VEL
LIN {X 0,Y 714.419,Z 707.31,A -85,B 0,C 180,E1 2901.139,E2 2901.139} C_VEL
LIN {X 0,Y 714.224,Z 707.31,A -85,B 0,C 180,E1 2905.112,E2 2905.112} C_VEL
LIN {X 0,Y 714.078,Z 707.31,A -85,B 0,C 180,E1 2910.621,E2 2910.621} C_VEL
LIN {X 0,Y 714.149,Z 707.31,A -85,B 0,C 180,E1 2916.454,E2 2916.454} C_VEL
LIN {X 0,Y 714.176,Z 707.31,A -85,B 0,C 180,E1 2921.133,E2 2921.133} C_VEL
LIN {X 0,Y 714.13,Z 707.31,A -85,B 0,C 180,E1 2926.18,E2 2926.18} C_VEL
LIN {X 0,Y 714.361,Z 707.31,A -85,B 0,C 180,E1 2932.035,E2 2932.035} C_VEL
LIN {X 0,Y 714.151,Z 707.463,A -85,B 0,C 180,E1 2936.516,E2 2936.516} C_VEL
LIN {X 0,Y 721.777,Z 725.345,A -85,B 0,C 180,E1 2937.089,E2 2937.089} C_VEL
LIN {X 0,Y 721.221,Z 773.814,A -85,B 0,C 180,E1 2937.91,E2 2937.91} C_VEL
LIN {X 0,Y 720.263,Z 817.857,A -85,B 0,C 180,E1 2939.181,E2 2939.181} C_VEL
LIN {X 0,Y 719.189,Z 859.17,A -85,B 0,C 180,E1 2940.879,E2 2940.879} C_VEL
LIN {X 0,Y 718.028,Z 899.821,A -85,B 0,C 180,E1 2943.112,E2 2943.112} C_VEL
LIN {X 0,Y 716.827,Z 937.832,A -85,B 0,C 180,E1 2945.83,E2 2945.83} C_VEL
LIN {X 0,Y 715.945,Z 971.249,A -85,B 0,C 180,E1 2948.911,E2 2948.911} C_VEL
LIN {X 0,Y 715.348,Z 999.539,A -85,B 0,C 180,E1 2952.284,E2 2952.284} C_VEL
LIN {X 0,Y 715.038,Z 1022.256,A -85,B 0,C 180,E1 2955.894,E2 2955.894} C_VEL
LIN {X 0,Y 714.817,Z 1038.758,A -85,B 0,C 180,E1 2959.619,E2 2959.619} C_VEL
LIN {X 0,Y 714.762,Z 1048.882,A -85,B 0,C 180,E1 2963.304,E2 2963.304} C_VEL
LIN {X 0,Y 714.714,Z 1052.912,A -85,B 0,C 180,E1 2966.354,E2 2966.354} C_VEL
LIN {X 0,Y 714.802,Z 1052.542,A -85,B 0,C 180,E1 2970.001,E2 2970.001} C_VEL
LIN {X 0,Y 714.837,Z 1046.636,A -85,B 0,C 180,E1 2973.647,E2 2973.647} C_VEL
LIN {X 0,Y 714.896,Z 1034.943,A -85,B 0,C 180,E1 2977.308,E2 2977.308} C_VEL
LIN {X 0,Y 715.077,Z 1016.742,A -85,B 0,C 180,E1 2980.996,E2 2980.996} C_VEL
LIN {X 0,Y 715.478,Z 993.539,A -85,B 0,C 180,E1 2984.411,E2 2984.411} C_VEL
LIN {X 0,Y 716.125,Z 966.203,A -85,B 0,C 180,E1 2987.51,E2 2987.51} C_VEL
LIN {X 0,Y 717.05,Z 932.612,A -85,B 0,C 180,E1 2990.49,E2 2990.49} C_VEL
LIN {X 0,Y 718.152,Z 895.194,A -85,B 0,C 180,E1 2993.082,E2 2993.082} C_VEL
LIN {X 0,Y 719.412,Z 852.71,A -85,B 0,C 180,E1 2995.332,E2 2995.332} C_VEL
LIN {X 0,Y 720.527,Z 807.25,A -85,B 0,C 180,E1 2997.088,E2 2997.088} C_VEL
LIN {X 0,Y 721.435,Z 760.901,A -85,B 0,C 180,E1 2998.275,E2 2998.275} C_VEL
LIN {X 0,Y 721.19,Z 723.621,A -85,B 0,C 180,E1 2998.869,E2 2998.869} C_VEL
LIN {X 0,Y 714.43,Z 707.31,A -85,B 0,C 180,E1 2999.4,E2 2999.4} C_VEL
LIN {X 0,Y 714.178,Z 707.31,A -85,B 0,C 180,E1 3004.954,E2 3004.954} C_VEL
LIN {X 0,Y 714.172,Z 707.31,A -85,B 0,C 180,E1 3010.19,E2 3010.19} C_VEL
LIN {X 0,Y 714.267,Z 707.31,A -85,B 0,C 180,E1 3015.56,E2 3015.56} C_VEL
LIN {X 0,Y 714.212,Z 707.31,A -85,B 0,C 180,E1 3020.464,E2 3020.464} C_VEL
LIN {X 0,Y 714.214,Z 707.31,A -85,B 0,C 180,E1 3025.843,E2 3025.843} C_VEL
LIN {X 0,Y 714.145,Z 707.31,A -85,B 0,C 180,E1 3030.785,E2 3030.785} C_VEL
LIN {X 0,Y 714.08,Z 707.31,A -85,B 0,C 180,E1 3035.859,E2 3035.859} C_VEL
LIN {X 0,Y 714.296,Z 707.31,A -85,B 0,C 180,E1 3040.155,E2 3040.155} C_VEL
LIN {X 0,Y 714.595,Z 707.31,A -85,B 0,C 180,E1 3046.508,E2 3046.508} C_VEL
LIN {X 0,Y 714.488,Z 707.31,A -85,B 0,C 180,E1 3051.861,E2 3051.861} C_VEL
LIN {X 0,Y 714.314,Z 707.31,A -85,B 0,C 180,E1 3056.349,E2 3056.349} C_VEL
LIN {X 0,Y 714.656,Z 707.31,A -85,B 0,C 180,E1 3061.213,E2 3061.213} C_VEL
LIN {X 0,Y 714.551,Z 707.31,A -85,B 0,C 180,E1 3067.652,E2 3067.652} C_VEL
LIN {X 0,Y 714.543,Z 707.31,A -85,B 0,C 180,E1 3070.38,E2 3070.38} C_VEL
LIN {X 0,Y 710.475,Z 707.31,A -85,B 0,C 180,E1 3071.745,E2 3071.745} C_VEL
LIN {X 0,Y 706.392,Z 707.31,A -85,B 0,C 180,E1 3073.126,E2 3073.126} C_VEL
LIN {X 0,Y 706.257,Z 707.31,A -85,B 0,C 180,E1 3078.772,E2 3078.772} C_VEL
LIN {X 0,Y 706.164,Z 707.31,A -85,B 0,C 180,E1 3084.06,E2 3084.06} C_VEL
LIN {X 0,Y 706.211,Z 707.31,A -85,B 0,C 180,E1 3088.383,E2 3088.383} C_VEL
LIN {X 0,Y 706.302,Z 707.31,A -85,B 0,C 180,E1 3093.199,E2 3093.199} C_VEL
LIN {X 0,Y 706.279,Z 707.31,A -85,B 0,C 180,E1 3098.476,E2 3098.476} C_VEL
LIN {X 0,Y 706.23,Z 707.31,A -85,B 0,C 180,E1 3103.361,E2 3103.361} C_VEL
LIN {X 0,Y 706.158,Z 707.31,A -85,B 0,C 180,E1 3108.681,E2 3108.681} C_VEL
LIN {X 0,Y 706.211,Z 707.31,A -85,B 0,C 180,E1 3113.07,E2 3113.07} C_VEL
LIN {X 0,Y 706.199,Z 708.023,A -85,B 0,C 180,E1 3117.82,E2 3117.82} C_VEL
LIN {X 0,Y 715.034,Z 728.116,A -85,B 0,C 180,E1 3118.497,E2 3118.497} C_VEL
LIN {X 0,Y 714.57,Z 790.773,A -85,B 0,C 180,E1 3119.354,E2 3119.354} C_VEL
LIN {X 0,Y 713.5,Z 838.859,A -85,B 0,C 180,E1 3120.604,E2 3120.604} C_VEL
LIN {X 0,Y 712.111,Z 885.108,A -85,B 0,C 180,E1 3122.428,E2 3122.428} C_VEL
LIN {X 0,Y 710.647,Z 929.002,A -85,B 0,C 180,E1 3124.827,E2 3124.827} C_VEL
LIN {X 0,Y 709.369,Z 967.512,A -85,B 0,C 180,E1 3127.602,E2 3127.602} C_VEL
LIN {X 0,Y 708.292,Z 1001.431,A -85,B 0,C 180,E1 3130.762,E2 3130.762} C_VEL
LIN {X 0,Y 707.603,Z 1030.187,A -85,B 0,C 180,E1 3134.247,E2 3134.247} C_VEL
LIN {X 0,Y 707.14,Z 1052.974,A -85,B 0,C 180,E1 3137.939,E2 3137.939} C_VEL
LIN {X 0,Y 706.887,Z 1069.161,A -85,B 0,C 180,E1 3141.679,E2 3141.679} C_VEL
LIN {X 0,Y 706.794,Z 1078.459,A -85,B 0,C 180,E1 3145.08,E2 3145.08} C_VEL
LIN {X 0,Y 706.746,Z 1083.169,A -85,B 0,C 180,E1 3148.771,E2 3148.771} C_VEL
LIN {X 0,Y 706.867,Z 1082.22,A -85,B 0,C 180,E1 3152.457,E2 3152.457} C_VEL
LIN {X 0,Y 706.776,Z 1077.195,A -85,B 0,C 180,E1 3155.536,E2 3155.536} C_VEL
LIN {X 0,Y 706.837,Z 1066.292,A -85,B 0,C 180,E1 3159.096,E2 3159.096} C_VEL
LIN {X 0,Y 707.089,Z 1051.279,A -85,B 0,C 180,E1 3162.375,E2 3162.375} C_VEL
LIN {X 0,Y 707.569,Z 1028.684,A -85,B 0,C 180,E1 3165.965,E2 3165.965} C_VEL
LIN {X 0,Y 708.28,Z 1000.328,A -85,B 0,C 180,E1 3169.36,E2 3169.36} C_VEL
LIN {X 0,Y 709.402,Z 966.231,A -85,B 0,C 180,E1 3172.505,E2 3172.505} C_VEL
LIN {X 0,Y 710.805,Z 926.578,A -85,B 0,C 180,E1 3175.321,E2 3175.321} C_VEL
LIN {X 0,Y 712.211,Z 885.132,A -85,B 0,C 180,E1 3177.566,E2 3177.566} C_VEL
LIN {X 0,Y 713.541,Z 840.721,A -85,B 0,C 180,E1 3179.327,E2 3179.327} C_VEL
LIN {X 0,Y 714.475,Z 798.399,A -85,B 0,C 180,E1 3180.48,E2 3180.48} C_VEL
LIN {X 0,Y 714.972,Z 754.752,A -85,B 0,C 180,E1 3181.199,E2 3181.199} C_VEL
LIN {X 0,Y 714.242,Z 725.144,A -85,B 0,C 180,E1 3181.577,E2 3181.577} C_VEL
LIN {X 0,Y 706.39,Z 707.31,A -85,B 0,C 180,E1 3182.255,E2 3182.255} C_VEL
LIN {X 0,Y 706.239,Z 707.31,A -85,B 0,C 180,E1 3187.451,E2 3187.451} C_VEL
LIN {X 0,Y 706.232,Z 707.31,A -85,B 0,C 180,E1 3191.696,E2 3191.696} C_VEL
LIN {X 0,Y 706.176,Z 707.31,A -85,B 0,C 180,E1 3196.853,E2 3196.853} C_VEL
LIN {X 0,Y 706.262,Z 707.31,A -85,B 0,C 180,E1 3201.523,E2 3201.523} C_VEL
LIN {X 0,Y 706.29,Z 707.31,A -85,B 0,C 180,E1 3206.8,E2 3206.8} C_VEL
LIN {X 0,Y 706.221,Z 707.31,A -85,B 0,C 180,E1 3211.834,E2 3211.834} C_VEL
LIN {X 0,Y 706.154,Z 707.31,A -85,B 0,C 180,E1 3215.94,E2 3215.94} C_VEL
LIN {X 0,Y 706.26,Z 707.31,A -85,B 0,C 180,E1 3221.228,E2 3221.228} C_VEL
LIN {X 0,Y 706.418,Z 707.31,A -85,B 0,C 180,E1 3226.354,E2 3226.354} C_VEL
LIN {X 0,Y 706.538,Z 707.31,A -85,B 0,C 180,E1 3231.367,E2 3231.367} C_VEL
LIN {X 0,Y 706.238,Z 707.31,A -85,B 0,C 180,E1 3235.079,E2 3235.079} C_VEL
LIN {X 0,Y 706.422,Z 707.31,A -85,B 0,C 180,E1 3240.002,E2 3240.002} C_VEL
LIN {X 0,Y 706.667,Z 707.31,A -85,B 0,C 180,E1 3244.923,E2 3244.923} C_VEL
LIN {X 0,Y 706.53,Z 707.31,A -85,B 0,C 180,E1 3251.132,E2 3251.132} C_VEL
LIN {X 0,Y 706.157,Z 707.31,A -85,B 0,C 180,E1 3256.201,E2 3256.201} C_VEL
LIN {X 0,Y 706.481,Z 707.31,A -85,B 0,C 180,E1 3261.388,E2 3261.388} C_VEL
LIN {X 0,Y 706.179,Z 707.31,A -85,B 0,C 180,E1 3265.674,E2 3265.674} C_VEL
LIN {X 0,Y 706.124,Z 707.31,A -85,B 0,C 180,E1 3271.004,E2 3271.004} C_VEL
LIN {X 0,Y 706.216,Z 707.31,A -85,B 0,C 180,E1 3275.408,E2 3275.408} C_VEL
LIN {X 0,Y 706.283,Z 707.31,A -85,B 0,C 180,E1 3280.069,E2 3280.069} C_VEL
LIN {X 0,Y 706.311,Z 707.31,A -85,B 0,C 180,E1 3285.076,E2 3285.076} C_VEL
LIN {X 0,Y 706.394,Z 707.31,A -85,B 0,C 180,E1 3290.563,E2 3290.563} C_VEL
LIN {X 0,Y 706.212,Z 707.31,A -85,B 0,C 180,E1 3294.631,E2 3294.631} C_VEL
LIN {X 0,Y 706.22,Z 707.838,A -85,B 0,C 180,E1 3296.127,E2 3296.127} C_VEL
LIN {X 0,Y 714.999,Z 729.157,A -85,B 0,C 180,E1 3296.814,E2 3296.814} C_VEL
LIN {X 0,Y 714.32,Z 776.192,A -85,B 0,C 180,E1 3297.644,E2 3297.644} C_VEL
LIN {X 0,Y 713.175,Z 822.35,A -85,B 0,C 180,E1 3299.03,E2 3299.03} C_VEL
LIN {X 0,Y 711.808,Z 865.039,A -85,B 0,C 180,E1 3300.872,E2 3300.872} C_VEL
LIN {X 0,Y 710.46,Z 904.87,A -85,B 0,C 180,E1 3303.166,E2 3303.166} C_VEL
LIN {X 0,Y 709.202,Z 940.758,A -85,B 0,C 180,E1 3305.831,E2 3305.831} C_VEL
LIN {X 0,Y 708.221,Z 972.512,A -85,B 0,C 180,E1 3308.834,E2 3308.834} C_VEL
LIN {X 0,Y 707.535,Z 1000.372,A -85,B 0,C 180,E1 3312.227,E2 3312.227} C_VEL
LIN {X 0,Y 707.172,Z 1022.122,A -85,B 0,C 180,E1 3315.734,E2 3315.734} C_VEL
LIN {X 0,Y 706.967,Z 1038.671,A -85,B 0,C 180,E1 3319.503,E2 3319.503} C_VEL
LIN {X 0,Y 706.875,Z 1048.838,A -85,B 0,C 180,E1 3323.229,E2 3323.229} C_VEL
LIN {X 0,Y 706.826,Z 1052.894,A -85,B 0,C 180,E1 3326.313,E2 3326.313} C_VEL
LIN {X 0,Y 706.929,Z 1052.561,A -85,B 0,C 180,E1 3330.001,E2 3330.001} C_VEL
LIN {X 0,Y 706.94,Z 1046.695,A -85,B 0,C 180,E1 3333.688,E2 3333.688} C_VEL
LIN {X 0,Y 706.992,Z 1035.031,A -85,B 0,C 180,E1 3337.39,E2 3337.39} C_VEL
LIN {X 0,Y 707.223,Z 1016.876,A -85,B 0,C 180,E1 3341.12,E2 3341.12} C_VEL
LIN {X 0,Y 707.694,Z 993.725,A -85,B 0,C 180,E1 3344.573,E2 3344.573} C_VEL
LIN {X 0,Y 708.455,Z 966.446,A -85,B 0,C 180,E1 3347.705,E2 3347.705} C_VEL
LIN {X 0,Y 709.504,Z 932.93,A -85,B 0,C 180,E1 3350.718,E2 3350.718} C_VEL
LIN {X 0,Y 710.789,Z 895.885,A -85,B 0,C 180,E1 3353.319,E2 3353.319} C_VEL
LIN {X 0,Y 712.259,Z 853.262,A -85,B 0,C 180,E1 3355.606,E2 3355.606} C_VEL
LIN {X 0,Y 713.543,Z 808.273,A -85,B 0,C 180,E1 3357.369,E2 3357.369} C_VEL
LIN {X 0,Y 714.567,Z 761.675,A -85,B 0,C 180,E1 3358.581,E2 3358.581} C_VEL
LIN {X 0,Y 714.496,Z 726.208,A -85,B 0,C 180,E1 3359.161,E2 3359.161} C_VEL
LIN {X 0,Y 706.439,Z 707.31,A -85,B 0,C 180,E1 3359.79,E2 3359.79} C_VEL
LIN {X 0,Y 706.263,Z 707.31,A -85,B 0,C 180,E1 3365.404,E2 3365.404} C_VEL
LIN {X 0,Y 706.274,Z 707.31,A -85,B 0,C 180,E1 3370.068,E2 3370.068} C_VEL
LIN {X 0,Y 706.323,Z 707.31,A -85,B 0,C 180,E1 3375.074,E2 3375.074} C_VEL
LIN {X 0,Y 706.297,Z 707.31,A -85,B 0,C 180,E1 3380.571,E2 3380.571} C_VEL
LIN {X 0,Y 706.299,Z 707.31,A -85,B 0,C 180,E1 3386.091,E2 3386.091} C_VEL
LIN {X 0,Y 706.278,Z 707.31,A -85,B 0,C 180,E1 3390.428,E2 3390.428} C_VEL
LIN {X 0,Y 706.292,Z 707.31,A -85,B 0,C 180,E1 3394.587,E2 3394.587} C_VEL
LIN {X 0,Y 706.394,Z 707.31,A -85,B 0,C 180,E1 3399.923,E2 3399.923} C_VEL
LIN {X 0,Y 706.648,Z 707.31,A -85,B 0,C 180,E1 3406.354,E2 3406.354} C_VEL
LIN {X 0,Y 706.563,Z 707.31,A -85,B 0,C 180,E1 3411.855,E2 3411.855} C_VEL
LIN {X 0,Y 706.43,Z 707.31,A -85,B 0,C 180,E1 3416.308,E2 3416.308} C_VEL
LIN {X 0,Y 706.743,Z 707.31,A -85,B 0,C 180,E1 3421.226,E2 3421.226} C_VEL
LIN {X 0,Y 706.714,Z 707.31,A -85,B 0,C 180,E1 3427.39,E2 3427.39} C_VEL
LIN {X 0,Y 706.445,Z 707.31,A -85,B 0,C 180,E1 3432.384,E2 3432.384} C_VEL
LIN {X 0,Y 706.392,Z 707.31,A -85,B 0,C 180,E1 3433.126,E2 3433.126} C_VEL
LIN {X 0,Y 702.399,Z 707.31,A -85,B 0,C 180,E1 3434.51,E2 3434.51} C_VEL
LIN {X 0,Y 698.324,Z 707.31,A -85,B 0,C 180,E1 3435.909,E2 3435.909} C_VEL
LIN {X 0,Y 698.339,Z 707.31,A -85,B 0,C 180,E1 3441.075,E2 3441.075} C_VEL
LIN {X 0,Y 698.409,Z 707.31,A -85,B 0,C 180,E1 3445.716,E2 3445.716} C_VEL
LIN {X 0,Y 698.462,Z 707.31,A -85,B 0,C 180,E1 3451.377,E2 3451.377} C_VEL
LIN {X 0,Y 698.345,Z 707.31,A -85,B 0,C 180,E1 3456.592,E2 3456.592} C_VEL
LIN {X 0,Y 698.284,Z 707.31,A -85,B 0,C 180,E1 3460.617,E2 3460.617} C_VEL
LIN {X 0,Y 698.269,Z 707.31,A -85,B 0,C 180,E1 3466.014,E2 3466.014} C_VEL
LIN {X 0,Y 698.353,Z 707.31,A -85,B 0,C 180,E1 3471.365,E2 3471.365} C_VEL
LIN {X 0,Y 698.252,Z 707.31,A -85,B 0,C 180,E1 3475.648,E2 3475.648} C_VEL
LIN {X 0,Y 698.252,Z 707.733,A -85,B 0,C 180,E1 3477.406,E2 3477.406} C_VEL
LIN {X 0,Y 708.189,Z 729.676,A -85,B 0,C 180,E1 3478.175,E2 3478.175} C_VEL
LIN {X 0,Y 707.772,Z 790.607,A -85,B 0,C 180,E1 3479.024,E2 3479.024} C_VEL
LIN {X 0,Y 706.569,Z 838.856,A -85,B 0,C 180,E1 3480.287,E2 3480.287} C_VEL
LIN {X 0,Y 704.966,Z 885.106,A -85,B 0,C 180,E1 3482.125,E2 3482.125} C_VEL
LIN {X 0,Y 703.381,Z 927.904,A -85,B 0,C 180,E1 3484.475,E2 3484.475} C_VEL
LIN {X 0,Y 701.904,Z 966.838,A -85,B 0,C 180,E1 3487.292,E2 3487.292} C_VEL
LIN {X 0,Y 700.639,Z 1000.905,A -85,B 0,C 180,E1 3490.485,E2 3490.485} C_VEL
LIN {X 0,Y 699.865,Z 1029.814,A -85,B 0,C 180,E1 3494.013,E2 3494.013} C_VEL
LIN {X 0,Y 699.281,Z 1052.975,A -85,B 0,C 180,E1 3497.801,E2 3497.801} C_VEL
LIN {X 0,Y 699.023,Z 1069.161,A -85,B 0,C 180,E1 3501.585,E2 3501.585} C_VEL
LIN {X 0,Y 698.906,Z 1078.459,A -85,B 0,C 180,E1 3505.024,E2 3505.024} C_VEL
LIN {X 0,Y 698.847,Z 1083.169,A -85,B 0,C 180,E1 3508.757,E2 3508.757} C_VEL
LIN {X 0,Y 698.966,Z 1082.219,A -85,B 0,C 180,E1 3512.485,E2 3512.485} C_VEL
LIN {X 0,Y 698.89,Z 1077.196,A -85,B 0,C 180,E1 3515.599,E2 3515.599} C_VEL
LIN {X 0,Y 698.977,Z 1066.571,A -85,B 0,C 180,E1 3519.123,E2 3519.123} C_VEL
LIN {X 0,Y 699.234,Z 1051.278,A -85,B 0,C 180,E1 3522.516,E2 3522.516} C_VEL
LIN {X 0,Y 699.8,Z 1028.473,A -85,B 0,C 180,E1 3526.175,E2 3526.175} C_VEL
LIN {X 0,Y 700.621,Z 999.93,A -85,B 0,C 180,E1 3529.622,E2 3529.622} C_VEL
LIN {X 0,Y 701.85,Z 966.833,A -85,B 0,C 180,E1 3532.71,E2 3532.71} C_VEL
LIN {X 0,Y 703.423,Z 927.928,A -85,B 0,C 180,E1 3535.522,E2 3535.522} C_VEL
LIN {X 0,Y 705.092,Z 885.13,A -85,B 0,C 180,E1 3537.869,E2 3537.869} C_VEL
LIN {X 0,Y 706.565,Z 840.718,A -85,B 0,C 180,E1 3539.645,E2 3539.645} C_VEL
LIN {X 0,Y 707.66,Z 798.32,A -85,B 0,C 180,E1 3540.807,E2 3540.807} C_VEL
LIN {X 0,Y 708.226,Z 752.399,A -85,B 0,C 180,E1 3541.558,E2 3541.558} C_VEL
LIN {X 0,Y 707.546,Z 727.958,A -85,B 0,C 180,E1 3541.877,E2 3541.877} C_VEL
LIN {X 0,Y 698.441,Z 707.31,A -85,B 0,C 180,E1 3542.627,E2 3542.627} C_VEL
LIN {X 0,Y 698.338,Z 707.31,A -85,B 0,C 180,E1 3547.416,E2 3547.416} C_VEL
LIN {X 0,Y 698.289,Z 707.31,A -85,B 0,C 180,E1 3552.455,E2 3552.455} C_VEL
LIN {X 0,Y 698.197,Z 707.31,A -85,B 0,C 180,E1 3557.717,E2 3557.717} C_VEL
LIN {X 0,Y 698.329,Z 707.31,A -85,B 0,C 180,E1 3562.587,E2 3562.587} C_VEL
LIN {X 0,Y 698.425,Z 707.31,A -85,B 0,C 180,E1 3567.799,E2 3567.799} C_VEL
LIN {X 0,Y 698.36,Z 707.31,A -85,B 0,C 180,E1 3572.894,E2 3572.894} C_VEL
LIN {X 0,Y 698.29,Z 707.31,A -85,B 0,C 180,E1 3578.353,E2 3578.353} C_VEL
LIN {X 0,Y 698.301,Z 707.31,A -85,B 0,C 180,E1 3583.616,E2 3583.616} C_VEL
LIN {X 0,Y 698.699,Z 707.31,A -85,B 0,C 180,E1 3588.746,E2 3588.746} C_VEL
LIN {X 0,Y 698.684,Z 707.31,A -85,B 0,C 180,E1 3593.777,E2 3593.777} C_VEL
LIN {X 0,Y 698.805,Z 707.31,A -85,B 0,C 180,E1 3598.76,E2 3598.76} C_VEL
LIN {X 0,Y 698.754,Z 707.31,A -85,B 0,C 180,E1 3604.979,E2 3604.979} C_VEL
LIN {X 0,Y 698.598,Z 707.31,A -85,B 0,C 180,E1 3611.26,E2 3611.26} C_VEL
LIN {X 0,Y 698.229,Z 707.31,A -85,B 0,C 180,E1 3616.39,E2 3616.39} C_VEL
LIN {X 0,Y 698.559,Z 707.31,A -85,B 0,C 180,E1 3621.643,E2 3621.643} C_VEL
LIN {X 0,Y 698.296,Z 707.31,A -85,B 0,C 180,E1 3625.726,E2 3625.726} C_VEL
LIN {X 0,Y 698.164,Z 707.31,A -85,B 0,C 180,E1 3631.397,E2 3631.397} C_VEL
LIN {X 0,Y 698.262,Z 707.31,A -85,B 0,C 180,E1 3636.584,E2 3636.584} C_VEL
LIN {X 0,Y 698.359,Z 707.31,A -85,B 0,C 180,E1 3640.618,E2 3640.618} C_VEL
LIN {X 0,Y 698.266,Z 707.31,A -85,B 0,C 180,E1 3646.016,E2 3646.016} C_VEL
LIN {X 0,Y 698.511,Z 707.31,A -85,B 0,C 180,E1 3651.356,E2 3651.356} C_VEL
LIN {X 0,Y 698.257,Z 707.31,A -85,B 0,C 180,E1 3655.694,E2 3655.694} C_VEL
LIN {X 0,Y 708.131,Z 729.789,A -85,B 0,C 180,E1 3656.486,E2 3656.486} C_VEL
LIN {X 0,Y 707.484,Z 776.118,A -85,B 0,C 180,E1 3657.318,E2 3657.318} C_VEL
LIN {X 0,Y 706.166,Z 821.154,A -85,B 0,C 180,E1 3658.671,E2 3658.671} C_VEL
LIN {X 0,Y 704.681,Z 862.835,A -85,B 0,C 180,E1 3660.461,E2 3660.461} C_VEL
LIN {X 0,Y 703.201,Z 902.76,A -85,B 0,C 180,E1 3662.75,E2 3662.75} C_VEL
LIN {X 0,Y 701.757,Z 938.881,A -85,B 0,C 180,E1 3665.42,E2 3665.42} C_VEL
LIN {X 0,Y 700.535,Z 972.025,A -85,B 0,C 180,E1 3668.561,E2 3668.561} C_VEL
LIN {X 0,Y 699.738,Z 1000.223,A -85,B 0,C 180,E1 3672.025,E2 3672.025} C_VEL
LIN {X 0,Y 699.33,Z 1021.988,A -85,B 0,C 180,E1 3675.571,E2 3675.571} C_VEL
LIN {X 0,Y 699.109,Z 1038.584,A -85,B 0,C 180,E1 3679.383,E2 3679.383} C_VEL
LIN {X 0,Y 698.98,Z 1048.793,A -85,B 0,C 180,E1 3683.152,E2 3683.152} C_VEL
LIN {X 0,Y 698.921,Z 1052.875,A -85,B 0,C 180,E1 3686.271,E2 3686.271} C_VEL
LIN {X 0,Y 699.027,Z 1052.58,A -85,B 0,C 180,E1 3690.001,E2 3690.001} C_VEL
LIN {X 0,Y 699.035,Z 1046.753,A -85,B 0,C 180,E1 3693.729,E2 3693.729} C_VEL
LIN {X 0,Y 699.097,Z 1035.117,A -85,B 0,C 180,E1 3697.474,E2 3697.474} C_VEL
LIN {X 0,Y 699.374,Z 1017.009,A -85,B 0,C 180,E1 3701.246,E2 3701.246} C_VEL
LIN {X 0,Y 699.911,Z 993.911,A -85,B 0,C 180,E1 3704.739,E2 3704.739} C_VEL
LIN {X 0,Y 700.801,Z 965.091,A -85,B 0,C 180,E1 3708.069,E2 3708.069} C_VEL
LIN {X 0,Y 702.04,Z 932.214,A -85,B 0,C 180,E1 3711.031,E2 3711.031} C_VEL
LIN {X 0,Y 703.494,Z 894.928,A -85,B 0,C 180,E1 3713.661,E2 3713.661} C_VEL
LIN {X 0,Y 705.13,Z 853.828,A -85,B 0,C 180,E1 3715.884,E2 3715.884} C_VEL
LIN {X 0,Y 706.596,Z 808.612,A -85,B 0,C 180,E1 3717.675,E2 3717.675} C_VEL
LIN {X 0,Y 707.768,Z 762.011,A -85,B 0,C 180,E1 3718.899,E2 3718.899} C_VEL
LIN {X 0,Y 707.616,Z 728.349,A -85,B 0,C 180,E1 3719.469,E2 3719.469} C_VEL
LIN {X 0,Y 698.473,Z 707.31,A -85,B 0,C 180,E1 3720.229,E2 3720.229} C_VEL
LIN {X 0,Y 698.297,Z 707.31,A -85,B 0,C 180,E1 3725.87,E2 3725.87} C_VEL
LIN {X 0,Y 698.311,Z 707.31,A -85,B 0,C 180,E1 3730.62,E2 3730.62} C_VEL
LIN {X 0,Y 698.35,Z 707.31,A -85,B 0,C 180,E1 3736.019,E2 3736.019} C_VEL
LIN {X 0,Y 698.385,Z 707.31,A -85,B 0,C 180,E1 3741.367,E2 3741.367} C_VEL
LIN {X 0,Y 698.382,Z 707.31,A -85,B 0,C 180,E1 3747.146,E2 3747.146} C_VEL
LIN {X 0,Y 698.316,Z 707.31,A -85,B 0,C 180,E1 3751.481,E2 3751.481} C_VEL
LIN {X 0,Y 698.303,Z 707.31,A -85,B 0,C 180,E1 3755.708,E2 3755.708} C_VEL
LIN {X 0,Y 698.371,Z 707.31,A -85,B 0,C 180,E1 3761.003,E2 3761.003} C_VEL
LIN {X 0,Y 698.713,Z 707.31,A -85,B 0,C 180,E1 3766.196,E2 3766.196} C_VEL
LIN {X 0,Y 698.658,Z 707.31,A -85,B 0,C 180,E1 3771.85,E2 3771.85} C_VEL
LIN {X 0,Y 698.537,Z 707.31,A -85,B 0,C 180,E1 3776.312,E2 3776.312} C_VEL
LIN {X 0,Y 698.83,Z 707.31,A -85,B 0,C 180,E1 3781.24,E2 3781.24} C_VEL
LIN {X 0,Y 698.791,Z 707.31,A -85,B 0,C 180,E1 3787.474,E2 3787.474} C_VEL
LIN {X 0,Y 698.528,Z 707.31,A -85,B 0,C 180,E1 3792.527,E2 3792.527} C_VEL
LIN {X 0,Y 698.324,Z 707.31,A -85,B 0,C 180,E1 3795.909,E2 3795.909} C_VEL
LIN {X 0,Y 694.285,Z 707.31,A -85,B 0,C 180,E1 3797.309,E2 3797.309} C_VEL
LIN {X 0,Y 690.381,Z 707.31,A -85,B 0,C 180,E1 3798.724,E2 3798.724} C_VEL
LIN {X 0,Y 690.301,Z 707.31,A -85,B 0,C 180,E1 3803.272,E2 3803.272} C_VEL
LIN {X 0,Y 690.438,Z 707.31,A -85,B 0,C 180,E1 3807.443,E2 3807.443} C_VEL
LIN {X 0,Y 690.555,Z 707.31,A -85,B 0,C 180,E1 3811.778,E2 3811.778} C_VEL
LIN {X 0,Y 690.43,Z 707.31,A -85,B 0,C 180,E1 3816.339,E2 3816.339} C_VEL
LIN {X 0,Y 690.295,Z 707.31,A -85,B 0,C 180,E1 3821.72,E2 3821.72} C_VEL
LIN {X 0,Y 690.287,Z 707.31,A -85,B 0,C 180,E1 3827.113,E2 3827.113} C_VEL
LIN {X 0,Y 690.408,Z 707.31,A -85,B 0,C 180,E1 3832.197,E2 3832.197} C_VEL
LIN {X 0,Y 690.33,Z 707.674,A -85,B 0,C 180,E1 3836.983,E2 3836.983} C_VEL
LIN {X 0,Y 701.586,Z 734.211,A -85,B 0,C 180,E1 3837.893,E2 3837.893} C_VEL
LIN {X 0,Y 700.97,Z 791.203,A -85,B 0,C 180,E1 3838.703,E2 3838.703} C_VEL
LIN {X 0,Y 699.666,Z 838.757,A -85,B 0,C 180,E1 3839.961,E2 3839.961} C_VEL
LIN {X 0,Y 697.941,Z 883.954,A -85,B 0,C 180,E1 3841.764,E2 3841.764} C_VEL
LIN {X 0,Y 696.038,Z 927.904,A -85,B 0,C 180,E1 3844.186,E2 3844.186} C_VEL
LIN {X 0,Y 694.412,Z 966.913,A -85,B 0,C 180,E1 3847.04,E2 3847.04} C_VEL
LIN {X 0,Y 692.93,Z 1001.561,A -85,B 0,C 180,E1 3850.332,E2 3850.332} C_VEL
LIN {X 0,Y 692.1,Z 1029.331,A -85,B 0,C 180,E1 3853.757,E2 3853.757} C_VEL
LIN {X 0,Y 691.445,Z 1052.976,A -85,B 0,C 180,E1 3857.661,E2 3857.661} C_VEL
LIN {X 0,Y 691.152,Z 1069.161,A -85,B 0,C 180,E1 3861.488,E2 3861.488} C_VEL
LIN {X 0,Y 691.011,Z 1078.46,A -85,B 0,C 180,E1 3864.967,E2 3864.967} C_VEL
LIN {X 0,Y 690.961,Z 1083.168,A -85,B 0,C 180,E1 3868.743,E2 3868.743} C_VEL
LIN {X 0,Y 691.094,Z 1082.219,A -85,B 0,C 180,E1 3872.513,E2 3872.513} C_VEL
LIN {X 0,Y 691.009,Z 1077.196,A -85,B 0,C 180,E1 3875.663,E2 3875.663} C_VEL
LIN {X 0,Y 691.1,Z 1066.086,A -85,B 0,C 180,E1 3879.362,E2 3879.362} C_VEL
LIN {X 0,Y 691.402,Z 1049.837,A -85,B 0,C 180,E1 3882.927,E2 3882.927} C_VEL
LIN {X 0,Y 691.998,Z 1028.233,A -85,B 0,C 180,E1 3886.395,E2 3886.395} C_VEL
LIN {X 0,Y 692.967,Z 999.42,A -85,B 0,C 180,E1 3889.901,E2 3889.901} C_VEL
LIN {X 0,Y 694.432,Z 964.867,A -85,B 0,C 180,E1 3893.128,E2 3893.128} C_VEL
LIN {X 0,Y 696.142,Z 926.795,A -85,B 0,C 180,E1 3895.88,E2 3895.88} C_VEL
LIN {X 0,Y 697.995,Z 884.019,A -85,B 0,C 180,E1 3898.231,E2 3898.231} C_VEL
LIN {X 0,Y 699.724,Z 837.987,A -85,B 0,C 180,E1 3900.064,E2 3900.064} C_VEL
LIN {X 0,Y 700.958,Z 791.952,A -85,B 0,C 180,E1 3901.28,E2 3901.28} C_VEL
LIN {X 0,Y 701.583,Z 740.406,A -85,B 0,C 180,E1 3902.033,E2 3902.033} C_VEL
LIN {X 0,Y 700.656,Z 730.036,A -85,B 0,C 180,E1 3902.204,E2 3902.204} C_VEL
LIN {X 0,Y 690.479,Z 707.31,A -85,B 0,C 180,E1 3903.049,E2 3903.049} C_VEL
LIN {X 0,Y 690.426,Z 707.31,A -85,B 0,C 180,E1 3907.92,E2 3907.92} C_VEL
LIN {X 0,Y 690.373,Z 707.31,A -85,B 0,C 180,E1 3913.588,E2 3913.588} C_VEL
LIN {X 0,Y 690.281,Z 707.31,A -85,B 0,C 180,E1 3918.81,E2 3918.81} C_VEL
LIN {X 0,Y 690.409,Z 707.31,A -85,B 0,C 180,E1 3924.303,E2 3924.303} C_VEL
LIN {X 0,Y 690.475,Z 707.31,A -85,B 0,C 180,E1 3929.686,E2 3929.686} C_VEL
LIN {X 0,Y 690.492,Z 707.31,A -85,B 0,C 180,E1 3934.132,E2 3934.132} C_VEL
LIN {X 0,Y 690.519,Z 707.31,A -85,B 0,C 180,E1 3939.446,E2 3939.446} C_VEL
LIN {X 0,Y 690.57,Z 707.31,A -85,B 0,C 180,E1 3944.913,E2 3944.913} C_VEL
LIN {X 0,Y 690.822,Z 707.31,A -85,B 0,C 180,E1 3949.895,E2 3949.895} C_VEL
LIN {X 0,Y 690.782,Z 707.31,A -85,B 0,C 180,E1 3953.705,E2 3953.705} C_VEL
LIN {X 0,Y 690.91,Z 707.31,A -85,B 0,C 180,E1 3958.746,E2 3958.746} C_VEL
LIN {X 0,Y 690.82,Z 707.31,A -85,B 0,C 180,E1 3965.036,E2 3965.036} C_VEL
LIN {X 0,Y 690.698,Z 707.31,A -85,B 0,C 180,E1 3971.391,E2 3971.391} C_VEL
LIN {X 0,Y 690.324,Z 707.31,A -85,B 0,C 180,E1 3976.583,E2 3976.583} C_VEL
LIN {X 0,Y 690.626,Z 707.31,A -85,B 0,C 180,E1 3981.904,E2 3981.904} C_VEL
LIN {X 0,Y 690.344,Z 707.31,A -85,B 0,C 180,E1 3986.044,E2 3986.044} C_VEL
LIN {X 0,Y 690.244,Z 707.31,A -85,B 0,C 180,E1 3991.106,E2 3991.106} C_VEL
LIN {X 0,Y 690.35,Z 707.31,A -85,B 0,C 180,E1 3996.35,E2 3996.35} C_VEL
LIN {X 0,Y 690.383,Z 707.31,A -85,B 0,C 180,E1 4001.73,E2 4001.73} C_VEL
LIN {X 0,Y 690.284,Z 707.31,A -85,B 0,C 180,E1 4007.114,E2 4007.114} C_VEL
LIN {X 0,Y 690.584,Z 707.31,A -85,B 0,C 180,E1 4012.186,E2 4012.186} C_VEL
LIN {X 0,Y 690.344,Z 707.31,A -85,B 0,C 180,E1 4015.283,E2 4015.283} C_VEL
LIN {X 0,Y 701.448,Z 734.167,A -85,B 0,C 180,E1 4016.213,E2 4016.213} C_VEL
LIN {X 0,Y 700.541,Z 778.866,A -85,B 0,C 180,E1 4017.056,E2 4017.056} C_VEL
LIN {X 0,Y 699.13,Z 824.017,A -85,B 0,C 180,E1 4018.454,E2 4018.454} C_VEL
LIN {X 0,Y 697.328,Z 868.623,A -85,B 0,C 180,E1 4020.448,E2 4020.448} C_VEL
LIN {X 0,Y 695.486,Z 911.315,A -85,B 0,C 180,E1 4023.039,E2 4023.039} C_VEL
LIN {X 0,Y 693.967,Z 947.937,A -85,B 0,C 180,E1 4025.951,E2 4025.951} C_VEL
LIN {X 0,Y 692.673,Z 981.061,A -85,B 0,C 180,E1 4029.361,E2 4029.361} C_VEL
LIN {X 0,Y 691.852,Z 1007.034,A -85,B 0,C 180,E1 4032.854,E2 4032.854} C_VEL
LIN {X 0,Y 691.324,Z 1028.169,A -85,B 0,C 180,E1 4036.694,E2 4036.694} C_VEL
LIN {X 0,Y 691.053,Z 1042.084,A -85,B 0,C 180,E1 4040.371,E2 4040.371} C_VEL
LIN {X 0,Y 691.059,Z 1049.954,A -85,B 0,C 180,E1 4043.706,E2 4043.706} C_VEL
LIN {X 0,Y 690.909,Z 1053.382,A -85,B 0,C 180,E1 4047.486,E2 4047.486} C_VEL
LIN {X 0,Y 690.989,Z 1051.289,A -85,B 0,C 180,E1 4051.257,E2 4051.257} C_VEL
LIN {X 0,Y 691.038,Z 1044.677,A -85,B 0,C 180,E1 4054.637,E2 4054.637} C_VEL
LIN {X 0,Y 691.14,Z 1032.601,A -85,B 0,C 180,E1 4058.194,E2 4058.194} C_VEL
LIN {X 0,Y 691.533,Z 1015.382,A -85,B 0,C 180,E1 4061.696,E2 4061.696} C_VEL
LIN {X 0,Y 692.282,Z 989.809,A -85,B 0,C 180,E1 4065.479,E2 4065.479} C_VEL
LIN {X 0,Y 693.473,Z 958.472,A -85,B 0,C 180,E1 4068.969,E2 4068.969} C_VEL
LIN {X 0,Y 694.923,Z 923.657,A -85,B 0,C 180,E1 4071.972,E2 4071.972} C_VEL
LIN {X 0,Y 696.767,Z 882.627,A -85,B 0,C 180,E1 4074.69,E2 4074.69} C_VEL
LIN {X 0,Y 698.626,Z 838.403,A -85,B 0,C 180,E1 4076.881,E2 4076.881} C_VEL
LIN {X 0,Y 700.161,Z 794.375,A -85,B 0,C 180,E1 4078.435,E2 4078.435} C_VEL
LIN {X 0,Y 701.275,Z 750.784,A -85,B 0,C 180,E1 4079.437,E2 4079.437} C_VEL
LIN {X 0,Y 700.794,Z 730.69,A -85,B 0,C 180,E1 4079.779,E2 4079.779} C_VEL
LIN {X 0,Y 690.502,Z 707.31,A -85,B 0,C 180,E1 4080.625,E2 4080.625} C_VEL
LIN {X 0,Y 690.38,Z 707.31,A -85,B 0,C 180,E1 4086.346,E2 4086.346} C_VEL
LIN {X 0,Y 690.292,Z 707.31,A -85,B 0,C 180,E1 4091.718,E2 4091.718} C_VEL
LIN {X 0,Y 690.4,Z 707.31,A -85,B 0,C 180,E1 4097.12,E2 4097.12} C_VEL
LIN {X 0,Y 690.418,Z 707.31,A -85,B 0,C 180,E1 4102.202,E2 4102.202} C_VEL
LIN {X 0,Y 690.427,Z 707.31,A -85,B 0,C 180,E1 4106.719,E2 4106.719} C_VEL
LIN {X 0,Y 690.43,Z 707.31,A -85,B 0,C 180,E1 4111.397,E2 4111.397} C_VEL
LIN {X 0,Y 690.397,Z 707.31,A -85,B 0,C 180,E1 4115.35,E2 4115.35} C_VEL
LIN {X 0,Y 690.458,Z 707.31,A -85,B 0,C 180,E1 4120.777,E2 4120.777} C_VEL
LIN {X 0,Y 690.763,Z 707.31,A -85,B 0,C 180,E1 4126.033,E2 4126.033} C_VEL
LIN {X 0,Y 690.83,Z 707.31,A -85,B 0,C 180,E1 4131.165,E2 4131.165} C_VEL
LIN {X 0,Y 690.642,Z 707.31,A -85,B 0,C 180,E1 4136.223,E2 4136.223} C_VEL
LIN {X 0,Y 690.935,Z 707.31,A -85,B 0,C 180,E1 4141.254,E2 4141.254} C_VEL
LIN {X 0,Y 690.872,Z 707.31,A -85,B 0,C 180,E1 4147.56,E2 4147.56} C_VEL
LIN {X 0,Y 690.608,Z 707.31,A -85,B 0,C 180,E1 4152.673,E2 4152.673} C_VEL
LIN {X 0,Y 690.36,Z 707.31,A -85,B 0,C 180,E1 4157.895,E2 4157.895} C_VEL
LIN {X 0,Y 690.381,Z 707.31,A -85,B 0,C 180,E1 4158.724,E2 4158.724} C_VEL
LIN {X 0,Y 686.489,Z 707.31,A -85,B 0,C 180,E1 4160.14,E2 4160.14} C_VEL
LIN {X 0,Y 682.435,Z 707.31,A -85,B 0,C 180,E1 4161.572,E2 4161.572} C_VEL
LIN {X 0,Y 682.532,Z 707.31,A -85,B 0,C 180,E1 4166.36,E2 4166.36} C_VEL
LIN {X 0,Y 682.578,Z 707.31,A -85,B 0,C 180,E1 4172.193,E2 4172.193} C_VEL
LIN {X 0,Y 682.477,Z 707.31,A -85,B 0,C 180,E1 4176.93,E2 4176.93} C_VEL
LIN {X 0,Y 682.416,Z 707.31,A -85,B 0,C 180,E1 4181.77,E2 4181.77} C_VEL
LIN {X 0,Y 682.386,Z 707.31,A -85,B 0,C 180,E1 4187.121,E2 4187.121} C_VEL
LIN {X 0,Y 682.434,Z 707.31,A -85,B 0,C 180,E1 4191.554,E2 4191.554} C_VEL
LIN {X 0,Y 682.402,Z 707.63,A -85,B 0,C 180,E1 4196.549,E2 4196.549} C_VEL
LIN {X 0,Y 694.887,Z 736.755,A -85,B 0,C 180,E1 4197.577,E2 4197.577} C_VEL
LIN {X 0,Y 694.208,Z 791.357,A -85,B 0,C 180,E1 4198.367,E2 4198.367} C_VEL
LIN {X 0,Y 692.769,Z 838.244,A -85,B 0,C 180,E1 4199.612,E2 4199.612} C_VEL
LIN {X 0,Y 690.824,Z 884.753,A -85,B 0,C 180,E1 4201.485,E2 4201.485} C_VEL
LIN {X 0,Y 688.776,Z 927.903,A -85,B 0,C 180,E1 4203.894,E2 4203.894} C_VEL
LIN {X 0,Y 686.936,Z 966.913,A -85,B 0,C 180,E1 4206.775,E2 4206.775} C_VEL
LIN {X 0,Y 685.35,Z 1000.392,A -85,B 0,C 180,E1 4209.972,E2 4209.972} C_VEL
LIN {X 0,Y 684.307,Z 1029.548,A -85,B 0,C 180,E1 4213.599,E2 4213.599} C_VEL
LIN {X 0,Y 683.606,Z 1053.108,A -85,B 0,C 180,E1 4217.545,E2 4217.545} C_VEL
LIN {X 0,Y 683.268,Z 1069.161,A -85,B 0,C 180,E1 4221.39,E2 4221.39} C_VEL
LIN {X 0,Y 683.129,Z 1078.459,A -85,B 0,C 180,E1 4224.909,E2 4224.909} C_VEL
LIN {X 0,Y 683.062,Z 1083.168,A -85,B 0,C 180,E1 4228.728,E2 4228.728} C_VEL
LIN {X 0,Y 683.193,Z 1082.218,A -85,B 0,C 180,E1 4232.542,E2 4232.542} C_VEL
LIN {X 0,Y 683.13,Z 1075.636,A -85,B 0,C 180,E1 4236.368,E2 4236.368} C_VEL
LIN {X 0,Y 683.22,Z 1064.73,A -85,B 0,C 180,E1 4239.846,E2 4239.846} C_VEL
LIN {X 0,Y 683.605,Z 1047.784,A -85,B 0,C 180,E1 4243.459,E2 4243.459} C_VEL
LIN {X 0,Y 684.268,Z 1026.117,A -85,B 0,C 180,E1 4246.877,E2 4246.877} C_VEL
LIN {X 0,Y 685.368,Z 998.307,A -85,B 0,C 180,E1 4250.248,E2 4250.248} C_VEL
LIN {X 0,Y 686.968,Z 964.868,A -85,B 0,C 180,E1 4253.394,E2 4253.394} C_VEL
LIN {X 0,Y 688.882,Z 925.993,A -85,B 0,C 180,E1 4256.225,E2 4256.225} C_VEL
LIN {X 0,Y 690.916,Z 883.694,A -85,B 0,C 180,E1 4258.562,E2 4258.562} C_VEL
LIN {X 0,Y 692.786,Z 838.282,A -85,B 0,C 180,E1 4260.386,E2 4260.386} C_VEL
LIN {X 0,Y 694.199,Z 791.71,A -85,B 0,C 180,E1 4261.625,E2 4261.625} C_VEL
LIN {X 0,Y 694.905,Z 737.987,A -85,B 0,C 180,E1 4262.408,E2 4262.408} C_VEL
LIN {X 0,Y 693.365,Z 731.451,A -85,B 0,C 180,E1 4262.567,E2 4262.567} C_VEL
LIN {X 0,Y 682.548,Z 707.31,A -85,B 0,C 180,E1 4263.479,E2 4263.479} C_VEL
LIN {X 0,Y 682.461,Z 707.31,A -85,B 0,C 180,E1 4269.002,E2 4269.002} C_VEL
LIN {X 0,Y 682.488,Z 707.31,A -85,B 0,C 180,E1 4274.726,E2 4274.726} C_VEL
LIN {X 0,Y 682.417,Z 707.31,A -85,B 0,C 180,E1 4279.914,E2 4279.914} C_VEL
LIN {X 0,Y 682.524,Z 707.31,A -85,B 0,C 180,E1 4285.235,E2 4285.235} C_VEL
LIN {X 0,Y 682.498,Z 707.31,A -85,B 0,C 180,E1 4290.762,E2 4290.762} C_VEL
LIN {X 0,Y 682.452,Z 707.31,A -85,B 0,C 180,E1 4295.561,E2 4295.561} C_VEL
LIN {X 0,Y 682.589,Z 707.31,A -85,B 0,C 180,E1 4300.551,E2 4300.551} C_VEL
LIN {X 0,Y 682.679,Z 707.31,A -85,B 0,C 180,E1 4305.869,E2 4305.869} C_VEL
LIN {X 0,Y 682.859,Z 707.31,A -85,B 0,C 180,E1 4311.066,E2 4311.066} C_VEL
LIN {X 0,Y 682.577,Z 707.31,A -85,B 0,C 180,E1 4314.908,E2 4314.908} C_VEL
LIN {X 0,Y 682.734,Z 707.31,A -85,B 0,C 180,E1 4320.002,E2 4320.002} C_VEL
LIN {X 0,Y 682.907,Z 707.31,A -85,B 0,C 180,E1 4325.095,E2 4325.095} C_VEL
LIN {X 0,Y 682.766,Z 707.31,A -85,B 0,C 180,E1 4331.525,E2 4331.525} C_VEL
LIN {X 0,Y 682.404,Z 707.31,A -85,B 0,C 180,E1 4336.782,E2 4336.782} C_VEL
LIN {X 0,Y 682.716,Z 707.31,A -85,B 0,C 180,E1 4342.171,E2 4342.171} C_VEL
LIN {X 0,Y 682.366,Z 707.31,A -85,B 0,C 180,E1 4347.801,E2 4347.801} C_VEL
LIN {X 0,Y 682.296,Z 707.31,A -85,B 0,C 180,E1 4352.437,E2 4352.437} C_VEL
LIN {X 0,Y 682.417,Z 707.31,A -85,B 0,C 180,E1 4356.926,E2 4356.926} C_VEL
LIN {X 0,Y 682.501,Z 707.31,A -85,B 0,C 180,E1 4361.77,E2 4361.77} C_VEL
